gfCNCPoint1[2427] = {X 506.1982, Y 15.6317, Z -1.3333, A 0.000, B 0.000, C 0.000 }
gfCNCPoint1[2428] = {X 505.5600, Y 16.3119, Z -1.3333, A 0.000, B 0.000, C 0.000 }
gfCNCPoint1[2429] = {X 505.5599, Y 40.8749, Z -1.3333, A 0.000, B 0.000, C 0.000 }
gfCNCPoint1[2430] = {X 506.2050, Y 41.5641, Z -1.3333, A 0.000, B 0.000, C 0.000 }
gfCNCPoint1[2431] = {X 506.6882, Y 42.3750, Z -1.3333, A 0.000, B 0.000, C 0.000 }
gfCNCPoint1[2432] = {X 506.9873, Y 43.2704, Z -1.3333, A 0.000, B 0.000, C 0.000 }
gfCNCPoint1[2433] = {X 507.0885, Y 44.2089, Z -1.3333, A 0.000, B 0.000, C 0.000 }
gfCNCPoint1[2434] = {X 507.0885, Y 45.0000, Z -1.3333, A 0.000, B 0.000, C 0.000 }
gfCNCPoint1[2435] = {X 506.9782, Y 45.9791, Z -1.3333, A 0.000, B 0.000, C 0.000 }
gfCNCPoint1[2436] = {X 506.6528, Y 46.9091, Z -1.3333, A 0.000, B 0.000, C 0.000 }
gfCNCPoint1[2437] = {X 506.1285, Y 47.7434, Z -1.3333, A 0.000, B 0.000, C 0.000 }
gfCNCPoint1[2438] = {X 505.4318, Y 48.4401, Z -1.3333, A 0.000, B 0.000, C 0.000 }
gfCNCPoint1[2439] = {X 504.5976, Y 48.9643, Z -1.3333, A 0.000, B 0.000, C 0.000 }
gfCNCPoint1[2440] = {X 503.6676, Y 49.2897, Z -1.3333, A 0.000, B 0.000, C 0.000 }
gfCNCPoint1[2441] = {X 502.6885, Y 49.4000, Z -1.3333, A 0.000, B 0.000, C 0.000 }
gfCNCPoint1[2442] = {X 496.2450, Y 49.4000, Z -1.3333, A 0.000, B 0.000, C 0.000 }
gfCNCPoint1[2443] = {X 495.2659, Y 49.2897, Z -1.3333, A 0.000, B 0.000, C 0.000 }
gfCNCPoint1[2444] = {X 494.3359, Y 48.9643, Z -1.3333, A 0.000, B 0.000, C 0.000 }
gfCNCPoint1[2445] = {X 493.5017, Y 48.4400, Z -1.3333, A 0.000, B 0.000, C 0.000 }
gfCNCPoint1[2446] = {X 492.8049, Y 47.7433, Z -1.3333, A 0.000, B 0.000, C 0.000 }
gfCNCPoint1[2447] = {X 492.2807, Y 46.9091, Z -1.3333, A 0.000, B 0.000, C 0.000 }
gfCNCPoint1[2448] = {X 491.9553, Y 45.9790, Z -1.3333, A 0.000, B 0.000, C 0.000 }
gfCNCPoint1[2449] = {X 491.8450, Y 44.9999, Z -1.3333, A 0.000, B 0.000, C 0.000 }
gfCNCPoint1[2450] = {X 491.8454, Y 44.1483, Z -1.3333, A 0.000, B 0.000, C 0.000 }
gfCNCPoint1[2451] = {X 491.9559, Y 43.2275, Z -1.3333, A 0.000, B 0.000, C 0.000 }
gfCNCPoint1[2452] = {X 492.2568, Y 42.3503, Z -1.3333, A 0.000, B 0.000, C 0.000 }
gfCNCPoint1[2453] = {X 492.7349, Y 41.5556, Z -1.3333, A 0.000, B 0.000, C 0.000 }
gfCNCPoint1[2454] = {X 493.3690, Y 40.8789, Z -1.3333, A 0.000, B 0.000, C 0.000 }
gfCNCPoint1[2455] = {X 493.3690, Y 34.5538, Z -1.3333, A 0.000, B 0.000, C 0.000 }
gfCNCPoint1[2456] = {X 490.7720, Y 34.5538, Z -1.3333, A 0.000, B 0.000, C 0.000 }
gfCNCPoint1[2457] = {X 486.5265, Y 42.8211, Z -1.3333, A 0.000, B 0.000, C 0.000 }
gfCNCPoint1[2458] = {X 486.6945, Y 43.5060, Z -1.3333, A 0.000, B 0.000, C 0.000 }
gfCNCPoint1[2459] = {X 486.7510, Y 44.2089, Z -1.3333, A 0.000, B 0.000, C 0.000 }
gfCNCPoint1[2460] = {X 486.7510, Y 45.0000, Z -1.3333, A 0.000, B 0.000, C 0.000 }
gfCNCPoint1[2461] = {X 486.6407, Y 45.9791, Z -1.3333, A 0.000, B 0.000, C 0.000 }
gfCNCPoint1[2462] = {X 486.3153, Y 46.9091, Z -1.3333, A 0.000, B 0.000, C 0.000 }
gfCNCPoint1[2463] = {X 485.7911, Y 47.7434, Z -1.3333, A 0.000, B 0.000, C 0.000 }
gfCNCPoint1[2464] = {X 485.0944, Y 48.4401, Z -1.3333, A 0.000, B 0.000, C 0.000 }
gfCNCPoint1[2465] = {X 484.2601, Y 48.9643, Z -1.3333, A 0.000, B 0.000, C 0.000 }
gfCNCPoint1[2466] = {X 483.3301, Y 49.2897, Z -1.3333, A 0.000, B 0.000, C 0.000 }
gfCNCPoint1[2467] = {X 482.3510, Y 49.4000, Z -1.3333, A 0.000, B 0.000, C 0.000 }
gfCNCPoint1[2468] = {X 480.2695, Y 49.4000, Z -1.3333, A 0.000, B 0.000, C 0.000 }
gfCNCPoint1[2469] = {X 480.2695, Y 49.8800, Z -1.3333, A 0.000, B 0.000, C 0.000 }
gfCNCPoint1[2470] = {X 481.4067, Y 50.7435, Z -1.3333, A 0.000, B 0.000, C 0.000 }
gfCNCPoint1[2471] = {X 482.4044, Y 51.7649, Z -1.3333, A 0.000, B 0.000, C 0.000 }
gfCNCPoint1[2472] = {X 483.2411, Y 52.9219, Z -1.3333, A 0.000, B 0.000, C 0.000 }
gfCNCPoint1[2473] = {X 483.8615, Y 54.1044, Z -1.3333, A 0.000, B 0.000, C 0.000 }
gfCNCPoint1[2474] = {X 484.3133, Y 55.3610, Z -1.3333, A 0.000, B 0.000, C 0.000 }
gfCNCPoint1[2475] = {X 484.5879, Y 56.6678, Z -1.3333, A 0.000, B 0.000, C 0.000 }
gfCNCPoint1[2476] = {X 484.6800, Y 58.0000, Z -1.3333, A 0.000, B 0.000, C 0.000 }
gfCNCPoint1[2477] = {X 484.6797, Y 59.0140, Z -1.3333, A 0.000, B 0.000, C 0.000 }
gfCNCPoint1[2478] = {X 484.5592, Y 60.4586, Z -1.3333, A 0.000, B 0.000, C 0.000 }
gfCNCPoint1[2479] = {X 484.2243, Y 61.8690, Z -1.3333, A 0.000, B 0.000, C 0.000 }
gfCNCPoint1[2480] = {X 483.6826, Y 63.2136, Z -1.3333, A 0.000, B 0.000, C 0.000 }
gfCNCPoint1[2481] = {X 482.9462, Y 64.4622, Z -1.3333, A 0.000, B 0.000, C 0.000 }
gfCNCPoint1[2482] = {X 482.0316, Y 65.5868, Z -1.3333, A 0.000, B 0.000, C 0.000 }
gfCNCPoint1[2483] = {X 480.9593, Y 66.5623, Z -1.3333, A 0.000, B 0.000, C 0.000 }
gfCNCPoint1[2484] = {X 480.9596, Y 89.4452, Z -1.3333, A 0.000, B 0.000, C 0.000 }
gfCNCPoint1[2485] = {X 482.0591, Y 90.4472, Z -1.3333, A 0.000, B 0.000, C 0.000 }
gfCNCPoint1[2486] = {X 482.9917, Y 91.6063, Z -1.3333, A 0.000, B 0.000, C 0.000 }
gfCNCPoint1[2487] = {X 483.7350, Y 92.8949, Z -1.3333, A 0.000, B 0.000, C 0.000 }
gfCNCPoint1[2488] = {X 507.6820, Y 92.8949, Z -1.3333, A 0.000, B 0.000, C 0.000 }
gfCNCPoint1[2489] = {X 507.6820, Y 95.2949, Z -1.3333, A 0.000, B 0.000, C 0.000 }
gfCNCPoint1[2490] = {X 595.2965, Y 95.2949, Z -1.3333, A 0.000, B 0.000, C 0.000 }
gfCNCPoint1[2491] = {X 595.2965, Y 54.2000, Z -1.3333, A 0.000, B 0.000, C 0.000 }
gfCNCPoint1[2492] = {X 593.5565, Y 54.2000, Z -1.3333, A 0.000, B 0.000, C 0.000 }
gfCNCPoint1[2493] = {X 592.2403, Y 54.1053, Z -1.3333, A 0.000, B 0.000, C 0.000 }
gfCNCPoint1[2494] = {X 590.9511, Y 53.8233, Z -1.3333, A 0.000, B 0.000, C 0.000 }
gfCNCPoint1[2495] = {X 589.7155, Y 53.3598, Z -1.3333, A 0.000, B 0.000, C 0.000 }
gfCNCPoint1[2496] = {X 588.5589, Y 52.7242, Z -1.3333, A 0.000, B 0.000, C 0.000 }
gfCNCPoint1[2497] = {X 587.5052, Y 51.9297, Z -1.3333, A 0.000, B 0.000, C 0.000 }
gfCNCPoint1[2498] = {X 586.4956, Y 52.6955, Z -1.3333, A 0.000, B 0.000, C 0.000 }
gfCNCPoint1[2499] = {X 585.3903, Y 53.3153, Z -1.3333, A 0.000, B 0.000, C 0.000 }
gfCNCPoint1[2500] = {X 584.1375, Y 53.7999, Z -1.3333, A 0.000, B 0.000, C 0.000 }
gfCNCPoint1[2501] = {X 582.8276, Y 54.0969, Z -1.3333, A 0.000, B 0.000, C 0.000 }
gfCNCPoint1[2502] = {X 581.4884, Y 54.1999, Z -1.3333, A 0.000, B 0.000, C 0.000 }
gfCNCPoint1[2503] = {X 580.1485, Y 54.1069, Z -1.3333, A 0.000, B 0.000, C 0.000 }
gfCNCPoint1[2504] = {X 578.8364, Y 53.8198, Z -1.3333, A 0.000, B 0.000, C 0.000 }
gfCNCPoint1[2505] = {X 577.5801, Y 53.3447, Z -1.3333, A 0.000, B 0.000, C 0.000 }
gfCNCPoint1[2506] = {X 576.4063, Y 52.6917, Z -1.3333, A 0.000, B 0.000, C 0.000 }
gfCNCPoint1[2507] = {X 575.3401, Y 51.8748, Z -1.3333, A 0.000, B 0.000, C 0.000 }
gfCNCPoint1[2508] = {X 574.2798, Y 52.6879, Z -1.3333, A 0.000, B 0.000, C 0.000 }
gfCNCPoint1[2509] = {X 573.1128, Y 53.3388, Z -1.3333, A 0.000, B 0.000, C 0.000 }
gfCNCPoint1[2510] = {X 571.8638, Y 53.8139, Z -1.3333, A 0.000, B 0.000, C 0.000 }
gfCNCPoint1[2511] = {X 570.5592, Y 54.1030, Z -1.3333, A 0.000, B 0.000, C 0.000 }
gfCNCPoint1[2512] = {X 569.2264, Y 54.2000, Z -1.3333, A 0.000, B 0.000, C 0.000 }
gfCNCPoint1[2513] = {X 562.4443, Y 54.2000, Z -1.3333, A 0.000, B 0.000, C 0.000 }
gfCNCPoint1[2514] = {X 561.0051, Y 54.0867, Z -1.3333, A 0.000, B 0.000, C 0.000 }
gfCNCPoint1[2515] = {X 559.6013, Y 53.7497, Z -1.3333, A 0.000, B 0.000, C 0.000 }
gfCNCPoint1[2516] = {X 558.2676, Y 53.1973, Z -1.3333, A 0.000, B 0.000, C 0.000 }
gfCNCPoint1[2517] = {X 557.0367, Y 52.4430, Z -1.3333, A 0.000, B 0.000, C 0.000 }
gfCNCPoint1[2518] = {X 555.9389, Y 51.5054, Z -1.3333, A 0.000, B 0.000, C 0.000 }
gfCNCPoint1[2519] = {X 555.0013, Y 50.4076, Z -1.3333, A 0.000, B 0.000, C 0.000 }
gfCNCPoint1[2520] = {X 554.2470, Y 49.1767, Z -1.3333, A 0.000, B 0.000, C 0.000 }
gfCNCPoint1[2521] = {X 553.6946, Y 47.8430, Z -1.3333, A 0.000, B 0.000, C 0.000 }
gfCNCPoint1[2522] = {X 553.3576, Y 46.4392, Z -1.3333, A 0.000, B 0.000, C 0.000 }
gfCNCPoint1[2523] = {X 553.2443, Y 45.0000, Z -1.3333, A 0.000, B 0.000, C 0.000 }
gfCNCPoint1[2524] = {X 553.2443, Y 44.0589, Z -1.3333, A 0.000, B 0.000, C 0.000 }
gfCNCPoint1[2525] = {X 553.3454, Y 42.7230, Z -1.3333, A 0.000, B 0.000, C 0.000 }
gfCNCPoint1[2526] = {X 553.6387, Y 41.4159, Z -1.3333, A 0.000, B 0.000, C 0.000 }
gfCNCPoint1[2527] = {X 554.1179, Y 40.1649, Z -1.3333, A 0.000, B 0.000, C 0.000 }
gfCNCPoint1[2528] = {X 554.7730, Y 38.9963, Z -1.3333, A 0.000, B 0.000, C 0.000 }
gfCNCPoint1[2529] = {X 554.7730, Y 11.0125, Z -1.3333, A 0.000, B 0.000, C 0.000 }
gfCNCPoint1[2530] = {X 554.1225, Y 9.8568, Z -1.3333, A 0.000, B 0.000, C 0.000 }
gfCNCPoint1[2531] = {X 553.6449, Y 8.6195, Z -1.3333, A 0.000, B 0.000, C 0.000 }
gfCNCPoint1[2532] = {X 553.3503, Y 7.3264, Z -1.3333, A 0.000, B 0.000, C 0.000 }
gfCNCPoint1[2533] = {X 553.2446, Y 6.0043, Z -1.3333, A 0.000, B 0.000, C 0.000 }
gfCNCPoint1[2534] = {X 553.2443, Y 5.0000, Z -1.3333, A 0.000, B 0.000, C 0.000 }
gfCNCPoint1[2535] = {X 553.2455, Y 4.8525, Z -1.3333, A 0.000, B 0.000, C 0.000 }
gfCNCPoint1[2536] = {X 553.2490, Y 4.7051, Z -1.3333, A 0.000, B 0.000, C 0.000 }
gfCNCPoint1[2537] = {X 365.1858, Y 4.7051, Z -1.3333, A 0.000, B 0.000, C 0.000 }
gfCNCPoint1[2538] = {X 365.5690, Y 5.1220, Z -1.3333, A 0.000, B 0.000, C 0.000 }
gfCNCPoint1[2539] = {X 365.9422, Y 5.5478, Z -1.3333, A 0.000, B 0.000, C 0.000 }
gfCNCPoint1[2540] = {X 367.0635, Y 6.9475, Z -1.3333, A 0.000, B 0.000, C 0.000 }
gfCNCPoint1[2541] = {X 368.0917, Y 8.4168, Z -1.3333, A 0.000, B 0.000, C 0.000 }
gfCNCPoint1[2542] = {X 369.3445, Y 10.5369, Z -1.3333, A 0.000, B 0.000, C 0.000 }
gfCNCPoint1[2543] = {X 370.4040, Y 12.7600, Z -1.3333, A 0.000, B 0.000, C 0.000 }
gfCNCPoint1[2544] = {X 371.2616, Y 15.0684, Z -1.3333, A 0.000, B 0.000, C 0.000 }
gfCNCPoint1[2545] = {X 371.9107, Y 17.4439, Z -1.3333, A 0.000, B 0.000, C 0.000 }
gfCNCPoint1[2546] = {X 372.3638, Y 19.8385, Z -1.3333, A 0.000, B 0.000, C 0.000 }
gfCNCPoint1[2547] = {X 372.6472, Y 22.2590, Z -1.3333, A 0.000, B 0.000, C 0.000 }
gfCNCPoint1[2548] = {X 372.7595, Y 24.6935, Z -1.3333, A 0.000, B 0.000, C 0.000 }
gfCNCPoint1[2549] = {X 372.7001, Y 27.1298, Z -1.3333, A 0.000, B 0.000, C 0.000 }
gfCNCPoint1[2550] = {X 372.4694, Y 29.5560, Z -1.3333, A 0.000, B 0.000, C 0.000 }
gfCNCPoint1[2551] = {X 372.0685, Y 31.9598, Z -1.3333, A 0.000, B 0.000, C 0.000 }
gfCNCPoint1[2552] = {X 371.4818, Y 34.3169, Z -1.3333, A 0.000, B 0.000, C 0.000 }
gfCNCPoint1[2553] = {X 370.6892, Y 36.6130, Z -1.3333, A 0.000, B 0.000, C 0.000 }
gfCNCPoint1[2554] = {X 369.6968, Y 38.8301, Z -1.3333, A 0.000, B 0.000, C 0.000 }
gfCNCPoint1[2555] = {X 368.5125, Y 40.9509, Z -1.3333, A 0.000, B 0.000, C 0.000 }
gfCNCPoint1[2556] = {X 367.1454, Y 42.9587, Z -1.3333, A 0.000, B 0.000, C 0.000 }
gfCNCPoint1[2557] = {X 365.7525, Y 44.6742, Z -1.3333, A 0.000, B 0.000, C 0.000 }
gfCNCPoint1[2558] = {X 364.2142, Y 46.2608, Z -1.3333, A 0.000, B 0.000, C 0.000 }
gfCNCPoint1[2559] = {X 362.5426, Y 47.7061, Z -1.3333, A 0.000, B 0.000, C 0.000 }
gfCNCPoint1[2560] = {X 360.7505, Y 48.9991, Z -1.3333, A 0.000, B 0.000, C 0.000 }
gfCNCPoint1[2561] = {X 358.8518, Y 50.1297, Z -1.3333, A 0.000, B 0.000, C 0.000 }
gfCNCPoint1[2562] = {X 356.6370, Y 51.1396, Z -1.3333, A 0.000, B 0.000, C 0.000 }
gfCNCPoint1[2563] = {X 354.3363, Y 51.9345, Z -1.3333, A 0.000, B 0.000, C 0.000 }
gfCNCPoint1[2564] = {X 351.9704, Y 52.5073, Z -1.3333, A 0.000, B 0.000, C 0.000 }
gfCNCPoint1[2565] = {X 349.5608, Y 52.8527, Z -1.3333, A 0.000, B 0.000, C 0.000 }
gfCNCPoint1[2566] = {X 347.1293, Y 52.9676, Z -1.3333, A 0.000, B 0.000, C 0.000 }
gfCNCPoint1[2567] = {X 344.8095, Y 52.9250, Z -1.3333, A 0.000, B 0.000, C 0.000 }
gfCNCPoint1[2568] = {X 342.5021, Y 52.6816, Z -1.3333, A 0.000, B 0.000, C 0.000 }
gfCNCPoint1[2569] = {X 340.2244, Y 52.2394, Z -1.3333, A 0.000, B 0.000, C 0.000 }
gfCNCPoint1[2570] = {X 337.9936, Y 51.6015, Z -1.3333, A 0.000, B 0.000, C 0.000 }
gfCNCPoint1[2571] = {X 335.8264, Y 50.7729, Z -1.3333, A 0.000, B 0.000, C 0.000 }
gfCNCPoint1[2572] = {X 333.7392, Y 49.7597, Z -1.3333, A 0.000, B 0.000, C 0.000 }
gfCNCPoint1[2573] = {X 332.8270, Y 49.2213, Z -1.3333, A 0.000, B 0.000, C 0.000 }
gfCNCPoint1[2574] = {X 331.9366, Y 48.6477, Z -1.3333, A 0.000, B 0.000, C 0.000 }
gfCNCPoint1[2575] = {X 331.3044, Y 48.2095, Z -1.3333, A 0.000, B 0.000, C 0.000 }
gfCNCPoint1[2576] = {X 330.6849, Y 47.7536, Z -1.3333, A 0.000, B 0.000, C 0.000 }
gfCNCPoint1[2577] = {X 329.2349, Y 49.6661, Z -1.3333, A 0.000, B 0.000, C 0.000 }
gfCNCPoint1[2578] = {X 328.8833, Y 49.3953, Z -1.3333, A 0.000, B 0.000, C 0.000 }
gfCNCPoint1[2579] = {X 328.5358, Y 49.1193, Z -1.3333, A 0.000, B 0.000, C 0.000 }
gfCNCPoint1[2580] = {X 328.1287, Y 49.0395, Z -1.3333, A 0.000, B 0.000, C 0.000 }
gfCNCPoint1[2581] = {X 327.7253, Y 48.9423, Z -1.3333, A 0.000, B 0.000, C 0.000 }
gfCNCPoint1[2582] = {X 328.4958, Y 49.2715, Z -1.3333, A 0.000, B 0.000, C 0.000 }
gfCNCPoint1[2583] = {X 329.2349, Y 49.6661, Z -1.3333, A 0.000, B 0.000, C 0.000 }
gfCNCPoint1[2584] = {X 330.6849, Y 47.7536, Z -1.3333, A 0.000, B 0.000, C 0.000 }
gfCNCPoint1[2585] = {X 330.1044, Y 47.3009, Z -1.3333, A 0.000, B 0.000, C 0.000 }
gfCNCPoint1[2586] = {X 329.5364, Y 46.8326, Z -1.3333, A 0.000, B 0.000, C 0.000 }
gfCNCPoint1[2587] = {X 328.9325, Y 46.7522, Z -1.3333, A 0.000, B 0.000, C 0.000 }
gfCNCPoint1[2588] = {X 328.3374, Y 46.6216, Z -1.3333, A 0.000, B 0.000, C 0.000 }
gfCNCPoint1[2589] = {X 327.9789, Y 46.5172, Z -1.3333, A 0.000, B 0.000, C 0.000 }
gfCNCPoint1[2590] = {X 327.6263, Y 46.3944, Z -1.3333, A 0.000, B 0.000, C 0.000 }
gfCNCPoint1[2591] = {X 326.7320, Y 45.9864, Z -1.3333, A 0.000, B 0.000, C 0.000 }
gfCNCPoint1[2592] = {X 325.9009, Y 45.4616, Z -1.3333, A 0.000, B 0.000, C 0.000 }
gfCNCPoint1[2593] = {X 325.1480, Y 44.8296, Z -1.3333, A 0.000, B 0.000, C 0.000 }
gfCNCPoint1[2594] = {X 324.5140, Y 44.2115, Z -1.3333, A 0.000, B 0.000, C 0.000 }
gfCNCPoint1[2595] = {X 324.0475, Y 43.7117, Z -1.3333, A 0.000, B 0.000, C 0.000 }
gfCNCPoint1[2596] = {X 323.6300, Y 43.1703, Z -1.3333, A 0.000, B 0.000, C 0.000 }
gfCNCPoint1[2597] = {X 319.6957, Y 45.9200, Z -1.3333, A 0.000, B 0.000, C 0.000 }
gfCNCPoint1[2598] = {X 319.4780, Y 45.5976, Z -1.3333, A 0.000, B 0.000, C 0.000 }
gfCNCPoint1[2599] = {X 319.2708, Y 45.2683, Z -1.3333, A 0.000, B 0.000, C 0.000 }
gfCNCPoint1[2600] = {X 319.2514, Y 45.5948, Z -1.3333, A 0.000, B 0.000, C 0.000 }
gfCNCPoint1[2601] = {X 319.2174, Y 45.9200, Z -1.3333, A 0.000, B 0.000, C 0.000 }
gfCNCPoint1[2602] = {X 319.6957, Y 45.9200, Z -1.3333, A 0.000, B 0.000, C 0.000 }
gfCNCPoint1[2603] = {X 321.6628, Y 44.5452, Z -1.3333, A 0.000, B 0.000, C 0.000 }
gfCNCPoint1[2604] = {X 321.4884, Y 44.2868, Z -1.3333, A 0.000, B 0.000, C 0.000 }
gfCNCPoint1[2605] = {X 321.3224, Y 44.0230, Z -1.3333, A 0.000, B 0.000, C 0.000 }
gfCNCPoint1[2606] = {X 320.6715, Y 42.7462, Z -1.3333, A 0.000, B 0.000, C 0.000 }
gfCNCPoint1[2607] = {X 320.2162, Y 41.3874, Z -1.3333, A 0.000, B 0.000, C 0.000 }
gfCNCPoint1[2608] = {X 319.9665, Y 39.9762, Z -1.3333, A 0.000, B 0.000, C 0.000 }
gfCNCPoint1[2609] = {X 319.9279, Y 38.5436, Z -1.3333, A 0.000, B 0.000, C 0.000 }
gfCNCPoint1[2610] = {X 320.1013, Y 37.1210, Z -1.3333, A 0.000, B 0.000, C 0.000 }
gfCNCPoint1[2611] = {X 320.4293, Y 35.8933, Z -1.3333, A 0.000, B 0.000, C 0.000 }
gfCNCPoint1[2612] = {X 320.9152, Y 34.7191, Z -1.3333, A 0.000, B 0.000, C 0.000 }
gfCNCPoint1[2613] = {X 321.5508, Y 33.6186, Z -1.3333, A 0.000, B 0.000, C 0.000 }
gfCNCPoint1[2614] = {X 324.1369, Y 29.7518, Z -1.3333, A 0.000, B 0.000, C 0.000 }
gfCNCPoint1[2615] = {X 320.1470, Y 27.0834, Z -1.3333, A 0.000, B 0.000, C 0.000 }
gfCNCPoint1[2616] = {X 321.7941, Y 24.6207, Z -1.3333, A 0.000, B 0.000, C 0.000 }
gfCNCPoint1[2617] = {X 321.9845, Y 24.3430, Z -1.3333, A 0.000, B 0.000, C 0.000 }
gfCNCPoint1[2618] = {X 322.1814, Y 24.0697, Z -1.3333, A 0.000, B 0.000, C 0.000 }
gfCNCPoint1[2619] = {X 321.5380, Y 23.0772, Z -1.3333, A 0.000, B 0.000, C 0.000 }
gfCNCPoint1[2620] = {X 320.9777, Y 22.0355, Z -1.3333, A 0.000, B 0.000, C 0.000 }
gfCNCPoint1[2621] = {X 320.1471, Y 20.3268, Z -1.3333, A 0.000, B 0.000, C 0.000 }
gfCNCPoint1[2622] = {X 320.1470, Y 27.0834, Z -1.3333, A 0.000, B 0.000, C 0.000 }
gfCNCPoint1[2623] = {X 322.1420, Y 28.4176, Z -1.3333, A 0.000, B 0.000, C 0.000 }
gfCNCPoint1[2624] = {X 323.7890, Y 25.9549, Z -1.3333, A 0.000, B 0.000, C 0.000 }
gfCNCPoint1[2625] = {X 324.5064, Y 24.9899, Z -1.3333, A 0.000, B 0.000, C 0.000 }
gfCNCPoint1[2626] = {X 325.3162, Y 24.1010, Z -1.3333, A 0.000, B 0.000, C 0.000 }
gfCNCPoint1[2627] = {X 324.4812, Y 23.1413, Z -1.3333, A 0.000, B 0.000, C 0.000 }
gfCNCPoint1[2628] = {X 323.7518, Y 22.0990, Z -1.3333, A 0.000, B 0.000, C 0.000 }
gfCNCPoint1[2629] = {X 323.1360, Y 20.9859, Z -1.3333, A 0.000, B 0.000, C 0.000 }
gfCNCPoint1[2630] = {X 319.6151, Y 13.7428, Z -1.3333, A 0.000, B 0.000, C 0.000 }
gfCNCPoint1[2631] = {X 319.4387, Y 13.3633, Z -1.3333, A 0.000, B 0.000, C 0.000 }
gfCNCPoint1[2632] = {X 319.2755, Y 12.9779, Z -1.3333, A 0.000, B 0.000, C 0.000 }
gfCNCPoint1[2633] = {X 319.2755, Y 13.0353, Z -1.3333, A 0.000, B 0.000, C 0.000 }
gfCNCPoint1[2634] = {X 319.1697, Y 14.2160, Z -1.3333, A 0.000, B 0.000, C 0.000 }
gfCNCPoint1[2635] = {X 318.8737, Y 15.3639, Z -1.3333, A 0.000, B 0.000, C 0.000 }
gfCNCPoint1[2636] = {X 318.3952, Y 16.4486, Z -1.3333, A 0.000, B 0.000, C 0.000 }
gfCNCPoint1[2637] = {X 317.7471, Y 17.4412, Z -1.3333, A 0.000, B 0.000, C 0.000 }
gfCNCPoint1[2638] = {X 317.7469, Y 36.6552, Z -1.3333, A 0.000, B 0.000, C 0.000 }
gfCNCPoint1[2639] = {X 318.1562, Y 35.1230, Z -1.3333, A 0.000, B 0.000, C 0.000 }
gfCNCPoint1[2640] = {X 318.7627, Y 33.6577, Z -1.3333, A 0.000, B 0.000, C 0.000 }
gfCNCPoint1[2641] = {X 319.5559, Y 32.2844, Z -1.3333, A 0.000, B 0.000, C 0.000 }
gfCNCPoint1[2642] = {X 322.1420, Y 28.4176, Z -1.3333, A 0.000, B 0.000, C 0.000 }
gfCNCPoint1[2643] = {X 324.1369, Y 29.7518, Z -1.3333, A 0.000, B 0.000, C 0.000 }
gfCNCPoint1[2644] = {X 325.7840, Y 27.2892, Z -1.3333, A 0.000, B 0.000, C 0.000 }
gfCNCPoint1[2645] = {X 326.3588, Y 26.5158, Z -1.3333, A 0.000, B 0.000, C 0.000 }
gfCNCPoint1[2646] = {X 327.0077, Y 25.8035, Z -1.3333, A 0.000, B 0.000, C 0.000 }
gfCNCPoint1[2647] = {X 328.0707, Y 24.8904, Z -1.3333, A 0.000, B 0.000, C 0.000 }
gfCNCPoint1[2648] = {X 329.2543, Y 24.1403, Z -1.3333, A 0.000, B 0.000, C 0.000 }
gfCNCPoint1[2649] = {X 328.0859, Y 23.3667, Z -1.3333, A 0.000, B 0.000, C 0.000 }
gfCNCPoint1[2650] = {X 327.0414, Y 22.4326, Z -1.3333, A 0.000, B 0.000, C 0.000 }
gfCNCPoint1[2651] = {X 326.3723, Y 21.6635, Z -1.3333, A 0.000, B 0.000, C 0.000 }
gfCNCPoint1[2652] = {X 325.7878, Y 20.8284, Z -1.3333, A 0.000, B 0.000, C 0.000 }
gfCNCPoint1[2653] = {X 325.2944, Y 19.9364, Z -1.3333, A 0.000, B 0.000, C 0.000 }
gfCNCPoint1[2654] = {X 321.7736, Y 12.6936, Z -1.3333, A 0.000, B 0.000, C 0.000 }
gfCNCPoint1[2655] = {X 321.6322, Y 12.3894, Z -1.3333, A 0.000, B 0.000, C 0.000 }
gfCNCPoint1[2656] = {X 321.5015, Y 12.0806, Z -1.3333, A 0.000, B 0.000, C 0.000 }
gfCNCPoint1[2657] = {X 321.1058, Y 10.8774, Z -1.3333, A 0.000, B 0.000, C 0.000 }
gfCNCPoint1[2658] = {X 320.8706, Y 9.6328, Z -1.3333, A 0.000, B 0.000, C 0.000 }
gfCNCPoint1[2659] = {X 320.7999, Y 8.3682, Z -1.3333, A 0.000, B 0.000, C 0.000 }
gfCNCPoint1[2660] = {X 320.8950, Y 7.1051, Z -1.3333, A 0.000, B 0.000, C 0.000 }
gfCNCPoint1[2661] = {X 298.7842, Y 7.1051, Z -1.3333, A 0.000, B 0.000, C 0.000 }
gfCNCPoint1[2662] = {X 298.7842, Y 9.5051, Z -1.3333, A 0.000, B 0.000, C 0.000 }
gfCNCPoint1[2663] = {X 297.8292, Y 9.5051, Z -1.3333, A 0.000, B 0.000, C 0.000 }
gfCNCPoint1[2664] = {X 298.1372, Y 10.4756, Z -1.3333, A 0.000, B 0.000, C 0.000 }
gfCNCPoint1[2665] = {X 298.3067, Y 11.4795, Z -1.3333, A 0.000, B 0.000, C 0.000 }
gfCNCPoint1[2666] = {X 298.4762, Y 10.4756, Z -1.3333, A 0.000, B 0.000, C 0.000 }
gfCNCPoint1[2667] = {X 298.7842, Y 9.5051, Z -1.3333, A 0.000, B 0.000, C 0.000 }
gfCNCPoint1[2668] = {X 298.7842, Y 7.1051, Z -1.3333, A 0.000, B 0.000, C 0.000 }
gfCNCPoint1[2669] = {X 233.3055, Y 7.1051, Z -1.3333, A 0.000, B 0.000, C 0.000 }
gfCNCPoint1[2670] = {X 233.3055, Y 11.9051, Z -1.3333, A 0.000, B 0.000, C 0.000 }
gfCNCPoint1[2671] = {X 233.1564, Y 11.9051, Z -1.3333, A 0.000, B 0.000, C 0.000 }
gfCNCPoint1[2672] = {X 233.1595, Y 12.0461, Z -1.3333, A 0.000, B 0.000, C 0.000 }
gfCNCPoint1[2673] = {X 233.1605, Y 12.1872, Z -1.3333, A 0.000, B 0.000, C 0.000 }
gfCNCPoint1[2674] = {X 233.2324, Y 12.0458, Z -1.3333, A 0.000, B 0.000, C 0.000 }
gfCNCPoint1[2675] = {X 233.3055, Y 11.9051, Z -1.3333, A 0.000, B 0.000, C 0.000 }
gfCNCPoint1[2676] = {X 233.3055, Y 9.5051, Z -1.3333, A 0.000, B 0.000, C 0.000 }
gfCNCPoint1[2677] = {X 230.2486, Y 9.5051, Z -1.3333, A 0.000, B 0.000, C 0.000 }
gfCNCPoint1[2678] = {X 230.6107, Y 10.7178, Z -1.3333, A 0.000, B 0.000, C 0.000 }
gfCNCPoint1[2679] = {X 230.7574, Y 11.9750, Z -1.3333, A 0.000, B 0.000, C 0.000 }
gfCNCPoint1[2680] = {X 230.7597, Y 12.0809, Z -1.3333, A 0.000, B 0.000, C 0.000 }
gfCNCPoint1[2681] = {X 230.7605, Y 12.1868, Z -1.3333, A 0.000, B 0.000, C 0.000 }
gfCNCPoint1[2682] = {X 230.7602, Y 13.0462, Z -1.3333, A 0.000, B 0.000, C 0.000 }
gfCNCPoint1[2683] = {X 230.6531, Y 14.2240, Z -1.3333, A 0.000, B 0.000, C 0.000 }
gfCNCPoint1[2684] = {X 230.3567, Y 15.3689, Z -1.3333, A 0.000, B 0.000, C 0.000 }
gfCNCPoint1[2685] = {X 229.8788, Y 16.4507, Z -1.3333, A 0.000, B 0.000, C 0.000 }
gfCNCPoint1[2686] = {X 229.2321, Y 17.4409, Z -1.3333, A 0.000, B 0.000, C 0.000 }
gfCNCPoint1[2687] = {X 229.2324, Y 25.8394, Z -1.3333, A 0.000, B 0.000, C 0.000 }
gfCNCPoint1[2688] = {X 231.6324, Y 25.8393, Z -1.3333, A 0.000, B 0.000, C 0.000 }
gfCNCPoint1[2689] = {X 231.6329, Y 38.9895, Z -1.3333, A 0.000, B 0.000, C 0.000 }
gfCNCPoint1[2690] = {X 231.6440, Y 39.0069, Z -1.3333, A 0.000, B 0.000, C 0.000 }
gfCNCPoint1[2691] = {X 232.3931, Y 37.9855, Z -1.3333, A 0.000, B 0.000, C 0.000 }
gfCNCPoint1[2692] = {X 233.2692, Y 37.0706, Z -1.3333, A 0.000, B 0.000, C 0.000 }
gfCNCPoint1[2693] = {X 234.2573, Y 36.2780, Z -1.3333, A 0.000, B 0.000, C 0.000 }
gfCNCPoint1[2694] = {X 235.5699, Y 33.7088, Z -1.3333, A 0.000, B 0.000, C 0.000 }
gfCNCPoint1[2695] = {X 234.4293, Y 32.2848, Z -1.3333, A 0.000, B 0.000, C 0.000 }
gfCNCPoint1[2696] = {X 233.4512, Y 30.7447, Z -1.3333, A 0.000, B 0.000, C 0.000 }
gfCNCPoint1[2697] = {X 232.6471, Y 29.1070, Z -1.3333, A 0.000, B 0.000, C 0.000 }
gfCNCPoint1[2698] = {X 232.0268, Y 27.3912, Z -1.3333, A 0.000, B 0.000, C 0.000 }
gfCNCPoint1[2699] = {X 231.8154, Y 26.6188, Z -1.3333, A 0.000, B 0.000, C 0.000 }
gfCNCPoint1[2700] = {X 231.6324, Y 25.8393, Z -1.3333, A 0.000, B 0.000, C 0.000 }
gfCNCPoint1[2701] = {X 229.2324, Y 25.8394, Z -1.3333, A 0.000, B 0.000, C 0.000 }
gfCNCPoint1[2702] = {X 229.2329, Y 39.7469, Z -1.3333, A 0.000, B 0.000, C 0.000 }
gfCNCPoint1[2703] = {X 229.4328, Y 40.0173, Z -1.3333, A 0.000, B 0.000, C 0.000 }
gfCNCPoint1[2704] = {X 229.6200, Y 40.2966, Z -1.3333, A 0.000, B 0.000, C 0.000 }
gfCNCPoint1[2705] = {X 230.1055, Y 41.1910, Z -1.3333, A 0.000, B 0.000, C 0.000 }
gfCNCPoint1[2706] = {X 230.4616, Y 42.1443, Z -1.3333, A 0.000, B 0.000, C 0.000 }
gfCNCPoint1[2707] = {X 230.6813, Y 43.1379, Z -1.3333, A 0.000, B 0.000, C 0.000 }
gfCNCPoint1[2708] = {X 230.7603, Y 44.1524, Z -1.3333, A 0.000, B 0.000, C 0.000 }
gfCNCPoint1[2709] = {X 230.7605, Y 45.0000, Z -1.3333, A 0.000, B 0.000, C 0.000 }
gfCNCPoint1[2710] = {X 230.7459, Y 45.4609, Z -1.3333, A 0.000, B 0.000, C 0.000 }
gfCNCPoint1[2711] = {X 230.7021, Y 45.9200, Z -1.3333, A 0.000, B 0.000, C 0.000 }
gfCNCPoint1[2712] = {X 232.5859, Y 45.9200, Z -1.3333, A 0.000, B 0.000, C 0.000 }
gfCNCPoint1[2713] = {X 232.5421, Y 45.4609, Z -1.3333, A 0.000, B 0.000, C 0.000 }
gfCNCPoint1[2714] = {X 232.5275, Y 45.0000, Z -1.3333, A 0.000, B 0.000, C 0.000 }
gfCNCPoint1[2715] = {X 232.5275, Y 44.2090, Z -1.3333, A 0.000, B 0.000, C 0.000 }
gfCNCPoint1[2716] = {X 232.6006, Y 43.1799, Z -1.3333, A 0.000, B 0.000, C 0.000 }
gfCNCPoint1[2717] = {X 232.8184, Y 42.1714, Z -1.3333, A 0.000, B 0.000, C 0.000 }
gfCNCPoint1[2718] = {X 233.1766, Y 41.2038, Z -1.3333, A 0.000, B 0.000, C 0.000 }
gfCNCPoint1[2719] = {X 233.6680, Y 40.2966, Z -1.3333, A 0.000, B 0.000, C 0.000 }
gfCNCPoint1[2720] = {X 234.3527, Y 39.3876, Z -1.3333, A 0.000, B 0.000, C 0.000 }
gfCNCPoint1[2721] = {X 235.1707, Y 38.5964, Z -1.3333, A 0.000, B 0.000, C 0.000 }
gfCNCPoint1[2722] = {X 236.1021, Y 37.9424, Z -1.3333, A 0.000, B 0.000, C 0.000 }
gfCNCPoint1[2723] = {X 238.5004, Y 33.2478, Z -1.3333, A 0.000, B 0.000, C 0.000 }
gfCNCPoint1[2724] = {X 237.3869, Y 32.1402, Z -1.3333, A 0.000, B 0.000, C 0.000 }
gfCNCPoint1[2725] = {X 236.4017, Y 30.9169, Z -1.3333, A 0.000, B 0.000, C 0.000 }
gfCNCPoint1[2726] = {X 235.5569, Y 29.5929, Z -1.3333, A 0.000, B 0.000, C 0.000 }
gfCNCPoint1[2727] = {X 234.8627, Y 28.1840, Z -1.3333, A 0.000, B 0.000, C 0.000 }
gfCNCPoint1[2728] = {X 234.3274, Y 26.7074, Z -1.3333, A 0.000, B 0.000, C 0.000 }
gfCNCPoint1[2729] = {X 234.1404, Y 26.0237, Z -1.3333, A 0.000, B 0.000, C 0.000 }
gfCNCPoint1[2730] = {X 233.9785, Y 25.3335, Z -1.3333, A 0.000, B 0.000, C 0.000 }
gfCNCPoint1[2731] = {X 233.6677, Y 23.4469, Z -1.3333, A 0.000, B 0.000, C 0.000 }
gfCNCPoint1[2732] = {X 233.5433, Y 21.5390, Z -1.3333, A 0.000, B 0.000, C 0.000 }
gfCNCPoint1[2733] = {X 233.6063, Y 19.6280, Z -1.3333, A 0.000, B 0.000, C 0.000 }
gfCNCPoint1[2734] = {X 233.8562, Y 17.7323, Z -1.3333, A 0.000, B 0.000, C 0.000 }
gfCNCPoint1[2735] = {X 234.2907, Y 15.8703, Z -1.3333, A 0.000, B 0.000, C 0.000 }
gfCNCPoint1[2736] = {X 234.7361, Y 14.5437, Z -1.3333, A 0.000, B 0.000, C 0.000 }
gfCNCPoint1[2737] = {X 235.3048, Y 13.2651, Z -1.3333, A 0.000, B 0.000, C 0.000 }
gfCNCPoint1[2738] = {X 235.3667, Y 13.1434, Z -1.3333, A 0.000, B 0.000, C 0.000 }
gfCNCPoint1[2739] = {X 235.4296, Y 13.0223, Z -1.3333, A 0.000, B 0.000, C 0.000 }
gfCNCPoint1[2740] = {X 236.1709, Y 11.7671, Z -1.3333, A 0.000, B 0.000, C 0.000 }
gfCNCPoint1[2741] = {X 237.0321, Y 10.5909, Z -1.3333, A 0.000, B 0.000, C 0.000 }
gfCNCPoint1[2742] = {X 238.0047, Y 9.5051, Z -1.3333, A 0.000, B 0.000, C 0.000 }
gfCNCPoint1[2743] = {X 233.3055, Y 9.5051, Z -1.3333, A 0.000, B 0.000, C 0.000 }
gfCNCPoint1[2744] = {X 233.3055, Y 7.1051, Z -1.3333, A 0.000, B 0.000, C 0.000 }
gfCNCPoint1[2745] = {X 207.3611, Y 7.1051, Z -1.3333, A 0.000, B 0.000, C 0.000 }
gfCNCPoint1[2746] = {X 207.3611, Y 11.9051, Z -1.3333, A 0.000, B 0.000, C 0.000 }
gfCNCPoint1[2747] = {X 205.8549, Y 11.9051, Z -1.3333, A 0.000, B 0.000, C 0.000 }
gfCNCPoint1[2748] = {X 206.6100, Y 13.3411, Z -1.3333, A 0.000, B 0.000, C 0.000 }
gfCNCPoint1[2749] = {X 207.2356, Y 14.8379, Z -1.3333, A 0.000, B 0.000, C 0.000 }
gfCNCPoint1[2750] = {X 207.7967, Y 16.7109, Z -1.3333, A 0.000, B 0.000, C 0.000 }
gfCNCPoint1[2751] = {X 208.1757, Y 18.6291, Z -1.3333, A 0.000, B 0.000, C 0.000 }
gfCNCPoint1[2752] = {X 208.3692, Y 20.5747, Z -1.3333, A 0.000, B 0.000, C 0.000 }
gfCNCPoint1[2753] = {X 208.3753, Y 22.5299, Z -1.3333, A 0.000, B 0.000, C 0.000 }
gfCNCPoint1[2754] = {X 208.1941, Y 24.4767, Z -1.3333, A 0.000, B 0.000, C 0.000 }
gfCNCPoint1[2755] = {X 207.8272, Y 26.3972, Z -1.3333, A 0.000, B 0.000, C 0.000 }
gfCNCPoint1[2756] = {X 207.3604, Y 28.0094, Z -1.3333, A 0.000, B 0.000, C 0.000 }
gfCNCPoint1[2757] = {X 206.7372, Y 29.5678, Z -1.3333, A 0.000, B 0.000, C 0.000 }
gfCNCPoint1[2758] = {X 205.9639, Y 31.0574, Z -1.3333, A 0.000, B 0.000, C 0.000 }
gfCNCPoint1[2759] = {X 206.0462, Y 31.2160, Z -1.3333, A 0.000, B 0.000, C 0.000 }
gfCNCPoint1[2760] = {X 206.1255, Y 31.3761, Z -1.3333, A 0.000, B 0.000, C 0.000 }
gfCNCPoint1[2761] = {X 208.8862, Y 37.0796, Z -1.3333, A 0.000, B 0.000, C 0.000 }
gfCNCPoint1[2762] = {X 208.8862, Y 18.1998, Z -1.3333, A 0.000, B 0.000, C 0.000 }
gfCNCPoint1[2763] = {X 208.2337, Y 17.0034, Z -1.3333, A 0.000, B 0.000, C 0.000 }
gfCNCPoint1[2764] = {X 207.7556, Y 15.7272, Z -1.3333, A 0.000, B 0.000, C 0.000 }
gfCNCPoint1[2765] = {X 207.4615, Y 14.3965, Z -1.3333, A 0.000, B 0.000, C 0.000 }
gfCNCPoint1[2766] = {X 207.3572, Y 13.0378, Z -1.3333, A 0.000, B 0.000, C 0.000 }
gfCNCPoint1[2767] = {X 207.3570, Y 12.1868, Z -1.3333, A 0.000, B 0.000, C 0.000 }
gfCNCPoint1[2768] = {X 207.3580, Y 12.0459, Z -1.3333, A 0.000, B 0.000, C 0.000 }
gfCNCPoint1[2769] = {X 207.3611, Y 11.9051, Z -1.3333, A 0.000, B 0.000, C 0.000 }
gfCNCPoint1[2770] = {X 207.3611, Y 9.5051, Z -1.3333, A 0.000, B 0.000, C 0.000 }
gfCNCPoint1[2771] = {X 200.9060, Y 9.5051, Z -1.3333, A 0.000, B 0.000, C 0.000 }
gfCNCPoint1[2772] = {X 201.9793, Y 10.6138, Z -1.3333, A 0.000, B 0.000, C 0.000 }
gfCNCPoint1[2773] = {X 202.9410, Y 11.8207, Z -1.3333, A 0.000, B 0.000, C 0.000 }
gfCNCPoint1[2774] = {X 203.7820, Y 13.1146, Z -1.3333, A 0.000, B 0.000, C 0.000 }
gfCNCPoint1[2775] = {X 204.4353, Y 14.3564, Z -1.3333, A 0.000, B 0.000, C 0.000 }
gfCNCPoint1[2776] = {X 204.9774, Y 15.6507, Z -1.3333, A 0.000, B 0.000, C 0.000 }
gfCNCPoint1[2777] = {X 205.5500, Y 17.6374, Z -1.3333, A 0.000, B 0.000, C 0.000 }
gfCNCPoint1[2778] = {X 205.8909, Y 19.6766, Z -1.3333, A 0.000, B 0.000, C 0.000 }
gfCNCPoint1[2779] = {X 205.9954, Y 21.7416, Z -1.3333, A 0.000, B 0.000, C 0.000 }
gfCNCPoint1[2780] = {X 205.8622, Y 23.8048, Z -1.3333, A 0.000, B 0.000, C 0.000 }
gfCNCPoint1[2781] = {X 205.4930, Y 25.8392, Z -1.3333, A 0.000, B 0.000, C 0.000 }
gfCNCPoint1[2782] = {X 205.0921, Y 27.2252, Z -1.3333, A 0.000, B 0.000, C 0.000 }
gfCNCPoint1[2783] = {X 204.5567, Y 28.5652, Z -1.3333, A 0.000, B 0.000, C 0.000 }
gfCNCPoint1[2784] = {X 203.8921, Y 29.8459, Z -1.3333, A 0.000, B 0.000, C 0.000 }
gfCNCPoint1[2785] = {X 203.1048, Y 31.0551, Z -1.3333, A 0.000, B 0.000, C 0.000 }
gfCNCPoint1[2786] = {X 203.5730, Y 31.7144, Z -1.3333, A 0.000, B 0.000, C 0.000 }
gfCNCPoint1[2787] = {X 203.9653, Y 32.4217, Z -1.3333, A 0.000, B 0.000, C 0.000 }
gfCNCPoint1[2788] = {X 206.9865, Y 38.6634, Z -1.3333, A 0.000, B 0.000, C 0.000 }
gfCNCPoint1[2789] = {X 207.4240, Y 39.8017, Z -1.3333, A 0.000, B 0.000, C 0.000 }
gfCNCPoint1[2790] = {X 207.6653, Y 40.9971, Z -1.3333, A 0.000, B 0.000, C 0.000 }
gfCNCPoint1[2791] = {X 207.7038, Y 42.2159, Z -1.3333, A 0.000, B 0.000, C 0.000 }
gfCNCPoint1[2792] = {X 207.5382, Y 43.4241, Z -1.3333, A 0.000, B 0.000, C 0.000 }
gfCNCPoint1[2793] = {X 207.1733, Y 44.5877, Z -1.3333, A 0.000, B 0.000, C 0.000 }
gfCNCPoint1[2794] = {X 206.6193, Y 45.6741, Z -1.3333, A 0.000, B 0.000, C 0.000 }
gfCNCPoint1[2795] = {X 205.8917, Y 46.6527, Z -1.3333, A 0.000, B 0.000, C 0.000 }
gfCNCPoint1[2796] = {X 205.0110, Y 47.4962, Z -1.3333, A 0.000, B 0.000, C 0.000 }
gfCNCPoint1[2797] = {X 204.4723, Y 47.9317, Z -1.3333, A 0.000, B 0.000, C 0.000 }
gfCNCPoint1[2798] = {X 203.5887, Y 48.5429, Z -1.3333, A 0.000, B 0.000, C 0.000 }
gfCNCPoint1[2799] = {X 202.6249, Y 49.0177, Z -1.3333, A 0.000, B 0.000, C 0.000 }
gfCNCPoint1[2800] = {X 201.4908, Y 49.3717, Z -1.3333, A 0.000, B 0.000, C 0.000 }
gfCNCPoint1[2801] = {X 200.3142, Y 49.5370, Z -1.3333, A 0.000, B 0.000, C 0.000 }
gfCNCPoint1[2802] = {X 199.1265, Y 49.5092, Z -1.3333, A 0.000, B 0.000, C 0.000 }
gfCNCPoint1[2803] = {X 198.4543, Y 49.8548, Z -1.3333, A 0.000, B 0.000, C 0.000 }
gfCNCPoint1[2804] = {X 197.7738, Y 50.1840, Z -1.3333, A 0.000, B 0.000, C 0.000 }
gfCNCPoint1[2805] = {X 199.8113, Y 54.5301, Z -1.3333, A 0.000, B 0.000, C 0.000 }
gfCNCPoint1[2806] = {X 197.9066, Y 55.3565, Z -1.3333, A 0.000, B 0.000, C 0.000 }
gfCNCPoint1[2807] = {X 195.9573, Y 56.0711, Z -1.3333, A 0.000, B 0.000, C 0.000 }
gfCNCPoint1[2808] = {X 195.3265, Y 56.2889, Z -1.3333, A 0.000, B 0.000, C 0.000 }
gfCNCPoint1[2809] = {X 195.3581, Y 56.6331, Z -1.3333, A 0.000, B 0.000, C 0.000 }
gfCNCPoint1[2810] = {X 195.3825, Y 56.9779, Z -1.3333, A 0.000, B 0.000, C 0.000 }
gfCNCPoint1[2811] = {X 199.6723, Y 61.6596, Z -1.3333, A 0.000, B 0.000, C 0.000 }
gfCNCPoint1[2812] = {X 199.5095, Y 60.3409, Z -1.3333, A 0.000, B 0.000, C 0.000 }
gfCNCPoint1[2813] = {X 199.4510, Y 59.0136, Z -1.3333, A 0.000, B 0.000, C 0.000 }
gfCNCPoint1[2814] = {X 199.4508, Y 58.0000, Z -1.3333, A 0.000, B 0.000, C 0.000 }
gfCNCPoint1[2815] = {X 199.5412, Y 56.2557, Z -1.3333, A 0.000, B 0.000, C 0.000 }
gfCNCPoint1[2816] = {X 199.8113, Y 54.5301, Z -1.3333, A 0.000, B 0.000, C 0.000 }
gfCNCPoint1[2817] = {X 198.7926, Y 52.3571, Z -1.3333, A 0.000, B 0.000, C 0.000 }
gfCNCPoint1[2818] = {X 197.0101, Y 53.1303, Z -1.3333, A 0.000, B 0.000, C 0.000 }
gfCNCPoint1[2819] = {X 195.1856, Y 53.7985, Z -1.3333, A 0.000, B 0.000, C 0.000 }
gfCNCPoint1[2820] = {X 194.5578, Y 54.0153, Z -1.3333, A 0.000, B 0.000, C 0.000 }
gfCNCPoint1[2821] = {X 193.5844, Y 54.3097, Z -1.3333, A 0.000, B 0.000, C 0.000 }
gfCNCPoint1[2822] = {X 192.6011, Y 54.5688, Z -1.3333, A 0.000, B 0.000, C 0.000 }
gfCNCPoint1[2823] = {X 192.9067, Y 56.2447, Z -1.3333, A 0.000, B 0.000, C 0.000 }
gfCNCPoint1[2824] = {X 193.0134, Y 57.9448, Z -1.3333, A 0.000, B 0.000, C 0.000 }
gfCNCPoint1[2825] = {X 210.3933, Y 76.9128, Z -1.3333, A 0.000, B 0.000, C 0.000 }
gfCNCPoint1[2826] = {X 212.1628, Y 75.2914, Z -1.3333, A 0.000, B 0.000, C 0.000 }
gfCNCPoint1[2827] = {X 215.1993, Y 78.6053, Z -1.3333, A 0.000, B 0.000, C 0.000 }
gfCNCPoint1[2828] = {X 218.3298, Y 76.5996, Z -1.3333, A 0.000, B 0.000, C 0.000 }
gfCNCPoint1[2829] = {X 216.9961, Y 76.0762, Z -1.3333, A 0.000, B 0.000, C 0.000 }
gfCNCPoint1[2830] = {X 216.3783, Y 75.8845, Z -1.3333, A 0.000, B 0.000, C 0.000 }
gfCNCPoint1[2831] = {X 215.7364, Y 75.8036, Z -1.3333, A 0.000, B 0.000, C 0.000 }
gfCNCPoint1[2832] = {X 213.9359, Y 75.6433, Z -1.3333, A 0.000, B 0.000, C 0.000 }
gfCNCPoint1[2833] = {X 212.1628, Y 75.2914, Z -1.3333, A 0.000, B 0.000, C 0.000 }
gfCNCPoint1[2834] = {X 210.3933, Y 76.9128, Z -1.3333, A 0.000, B 0.000, C 0.000 }
gfCNCPoint1[2835] = {X 214.7938, Y 81.7153, Z -1.3333, A 0.000, B 0.000, C 0.000 }
gfCNCPoint1[2836] = {X 223.5843, Y 76.0836, Z -1.3333, A 0.000, B 0.000, C 0.000 }
gfCNCPoint1[2837] = {X 217.8854, Y 73.8470, Z -1.3333, A 0.000, B 0.000, C 0.000 }
gfCNCPoint1[2838] = {X 216.8736, Y 73.5361, Z -1.3333, A 0.000, B 0.000, C 0.000 }
gfCNCPoint1[2839] = {X 215.8232, Y 73.4052, Z -1.3333, A 0.000, B 0.000, C 0.000 }
gfCNCPoint1[2840] = {X 214.2776, Y 73.2678, Z -1.3333, A 0.000, B 0.000, C 0.000 }
gfCNCPoint1[2841] = {X 212.7554, Y 72.9657, Z -1.3333, A 0.000, B 0.000, C 0.000 }
gfCNCPoint1[2842] = {X 211.1566, Y 72.4581, Z -1.3333, A 0.000, B 0.000, C 0.000 }
gfCNCPoint1[2843] = {X 209.6273, Y 71.7689, Z -1.3333, A 0.000, B 0.000, C 0.000 }
gfCNCPoint1[2844] = {X 208.1879, Y 70.9075, Z -1.3333, A 0.000, B 0.000, C 0.000 }
gfCNCPoint1[2845] = {X 206.8577, Y 69.8854, Z -1.3333, A 0.000, B 0.000, C 0.000 }
gfCNCPoint1[2846] = {X 205.6547, Y 68.7163, Z -1.3333, A 0.000, B 0.000, C 0.000 }
gfCNCPoint1[2847] = {X 204.5950, Y 67.4159, Z -1.3333, A 0.000, B 0.000, C 0.000 }
gfCNCPoint1[2848] = {X 203.6928, Y 66.0018, Z -1.3333, A 0.000, B 0.000, C 0.000 }
gfCNCPoint1[2849] = {X 202.9602, Y 64.4927, Z -1.3333, A 0.000, B 0.000, C 0.000 }
gfCNCPoint1[2850] = {X 202.4071, Y 62.9091, Z -1.3333, A 0.000, B 0.000, C 0.000 }
gfCNCPoint1[2851] = {X 202.0408, Y 61.2721, Z -1.3333, A 0.000, B 0.000, C 0.000 }
gfCNCPoint1[2852] = {X 201.9014, Y 60.1434, Z -1.3333, A 0.000, B 0.000, C 0.000 }
gfCNCPoint1[2853] = {X 201.8510, Y 59.0073, Z -1.3333, A 0.000, B 0.000, C 0.000 }
gfCNCPoint1[2854] = {X 201.8508, Y 58.0000, Z -1.3333, A 0.000, B 0.000, C 0.000 }
gfCNCPoint1[2855] = {X 201.9283, Y 56.5037, Z -1.3333, A 0.000, B 0.000, C 0.000 }
gfCNCPoint1[2856] = {X 202.1600, Y 55.0235, Z -1.3333, A 0.000, B 0.000, C 0.000 }
gfCNCPoint1[2857] = {X 202.4969, Y 53.7228, Z -1.3333, A 0.000, B 0.000, C 0.000 }
gfCNCPoint1[2858] = {X 202.9529, Y 52.4590, Z -1.3333, A 0.000, B 0.000, C 0.000 }
gfCNCPoint1[2859] = {X 203.5241, Y 51.2429, Z -1.3333, A 0.000, B 0.000, C 0.000 }
gfCNCPoint1[2860] = {X 202.2650, Y 51.6541, Z -1.3333, A 0.000, B 0.000, C 0.000 }
gfCNCPoint1[2861] = {X 200.9616, Y 51.8900, Z -1.3333, A 0.000, B 0.000, C 0.000 }
gfCNCPoint1[2862] = {X 199.6382, Y 51.9460, Z -1.3333, A 0.000, B 0.000, C 0.000 }
gfCNCPoint1[2863] = {X 199.2168, Y 52.1545, Z -1.3333, A 0.000, B 0.000, C 0.000 }
gfCNCPoint1[2864] = {X 198.7926, Y 52.3571, Z -1.3333, A 0.000, B 0.000, C 0.000 }
gfCNCPoint1[2865] = {X 197.7738, Y 50.1840, Z -1.3333, A 0.000, B 0.000, C 0.000 }
gfCNCPoint1[2866] = {X 196.1132, Y 50.9041, Z -1.3333, A 0.000, B 0.000, C 0.000 }
gfCNCPoint1[2867] = {X 194.4134, Y 51.5260, Z -1.3333, A 0.000, B 0.000, C 0.000 }
gfCNCPoint1[2868] = {X 193.8217, Y 51.7310, Z -1.3333, A 0.000, B 0.000, C 0.000 }
gfCNCPoint1[2869] = {X 192.9311, Y 52.0003, Z -1.3333, A 0.000, B 0.000, C 0.000 }
gfCNCPoint1[2870] = {X 192.0315, Y 52.2374, Z -1.3333, A 0.000, B 0.000, C 0.000 }
gfCNCPoint1[2871] = {X 190.7254, Y 52.5209, Z -1.3333, A 0.000, B 0.000, C 0.000 }
gfCNCPoint1[2872] = {X 189.4065, Y 52.7364, Z -1.3333, A 0.000, B 0.000, C 0.000 }
gfCNCPoint1[2873] = {X 189.9015, Y 53.9141, Z -1.3333, A 0.000, B 0.000, C 0.000 }
gfCNCPoint1[2874] = {X 190.2695, Y 55.1375, Z -1.3333, A 0.000, B 0.000, C 0.000 }
gfCNCPoint1[2875] = {X 190.5272, Y 56.5585, Z -1.3333, A 0.000, B 0.000, C 0.000 }
gfCNCPoint1[2876] = {X 190.6135, Y 58.0000, Z -1.3333, A 0.000, B 0.000, C 0.000 }
gfCNCPoint1[2877] = {X 190.6132, Y 58.8779, Z -1.3333, A 0.000, B 0.000, C 0.000 }
gfCNCPoint1[2878] = {X 214.3883, Y 84.8254, Z -1.3333, A 0.000, B 0.000, C 0.000 }
gfCNCPoint1[2879] = {X 228.8388, Y 75.5676, Z -1.3333, A 0.000, B 0.000, C 0.000 }
gfCNCPoint1[2880] = {X 218.7726, Y 71.6170, Z -1.3333, A 0.000, B 0.000, C 0.000 }
gfCNCPoint1[2881] = {X 217.8439, Y 71.3035, Z -1.3333, A 0.000, B 0.000, C 0.000 }
gfCNCPoint1[2882] = {X 216.8852, Y 71.0992, Z -1.3333, A 0.000, B 0.000, C 0.000 }
gfCNCPoint1[2883] = {X 215.9094, Y 71.0067, Z -1.3333, A 0.000, B 0.000, C 0.000 }
gfCNCPoint1[2884] = {X 214.2392, Y 70.8316, Z -1.3333, A 0.000, B 0.000, C 0.000 }
gfCNCPoint1[2885] = {X 212.6095, Y 70.4266, Z -1.3333, A 0.000, B 0.000, C 0.000 }
gfCNCPoint1[2886] = {X 211.0517, Y 69.7995, Z -1.3333, A 0.000, B 0.000, C 0.000 }
gfCNCPoint1[2887] = {X 209.5959, Y 68.9624, Z -1.3333, A 0.000, B 0.000, C 0.000 }
gfCNCPoint1[2888] = {X 208.2702, Y 67.9315, Z -1.3333, A 0.000, B 0.000, C 0.000 }
gfCNCPoint1[2889] = {X 207.1004, Y 66.7267, Z -1.3333, A 0.000, B 0.000, C 0.000 }
gfCNCPoint1[2890] = {X 206.1089, Y 65.3714, Z -1.3333, A 0.000, B 0.000, C 0.000 }
gfCNCPoint1[2891] = {X 205.3149, Y 63.8916, Z -1.3333, A 0.000, B 0.000, C 0.000 }
gfCNCPoint1[2892] = {X 204.7339, Y 62.3160, Z -1.3333, A 0.000, B 0.000, C 0.000 }
gfCNCPoint1[2893] = {X 204.3769, Y 60.6751, Z -1.3333, A 0.000, B 0.000, C 0.000 }
gfCNCPoint1[2894] = {X 204.2510, Y 59.0005, Z -1.3333, A 0.000, B 0.000, C 0.000 }
gfCNCPoint1[2895] = {X 204.2508, Y 58.0000, Z -1.3333, A 0.000, B 0.000, C 0.000 }
gfCNCPoint1[2896] = {X 204.3397, Y 56.5374, Z -1.3333, A 0.000, B 0.000, C 0.000 }
gfCNCPoint1[2897] = {X 204.6050, Y 55.0963, Z -1.3333, A 0.000, B 0.000, C 0.000 }
gfCNCPoint1[2898] = {X 205.0428, Y 53.6979, Z -1.3333, A 0.000, B 0.000, C 0.000 }
gfCNCPoint1[2899] = {X 205.6468, Y 52.3629, Z -1.3333, A 0.000, B 0.000, C 0.000 }
gfCNCPoint1[2900] = {X 206.5302, Y 50.9378, Z -1.3333, A 0.000, B 0.000, C 0.000 }
gfCNCPoint1[2901] = {X 207.6025, Y 49.6488, Z -1.3333, A 0.000, B 0.000, C 0.000 }
gfCNCPoint1[2902] = {X 208.8430, Y 48.5206, Z -1.3333, A 0.000, B 0.000, C 0.000 }
gfCNCPoint1[2903] = {X 210.2277, Y 47.5751, Z -1.3333, A 0.000, B 0.000, C 0.000 }
gfCNCPoint1[2904] = {X 209.8801, Y 46.3328, Z -1.3333, A 0.000, B 0.000, C 0.000 }
gfCNCPoint1[2905] = {X 209.7572, Y 45.0487, Z -1.3333, A 0.000, B 0.000, C 0.000 }
gfCNCPoint1[2906] = {X 209.7570, Y 44.2008, Z -1.3333, A 0.000, B 0.000, C 0.000 }
gfCNCPoint1[2907] = {X 209.8559, Y 43.0097, Z -1.3333, A 0.000, B 0.000, C 0.000 }
gfCNCPoint1[2908] = {X 210.1500, Y 41.8513, Z -1.3333, A 0.000, B 0.000, C 0.000 }
gfCNCPoint1[2909] = {X 210.6312, Y 40.7572, Z -1.3333, A 0.000, B 0.000, C 0.000 }
gfCNCPoint1[2910] = {X 211.2862, Y 39.7575, Z -1.3333, A 0.000, B 0.000, C 0.000 }
gfCNCPoint1[2911] = {X 211.2862, Y 37.0796, Z -1.3333, A 0.000, B 0.000, C 0.000 }
gfCNCPoint1[2912] = {X 211.2860, Y 17.4416, Z -1.3333, A 0.000, B 0.000, C 0.000 }
gfCNCPoint1[2913] = {X 210.6370, Y 16.4476, Z -1.3333, A 0.000, B 0.000, C 0.000 }
gfCNCPoint1[2914] = {X 210.1582, Y 15.3613, Z -1.3333, A 0.000, B 0.000, C 0.000 }
gfCNCPoint1[2915] = {X 209.8623, Y 14.2116, Z -1.3333, A 0.000, B 0.000, C 0.000 }
gfCNCPoint1[2916] = {X 209.7572, Y 13.0291, Z -1.3333, A 0.000, B 0.000, C 0.000 }
gfCNCPoint1[2917] = {X 209.7570, Y 12.1868, Z -1.3333, A 0.000, B 0.000, C 0.000 }
gfCNCPoint1[2918] = {X 209.7578, Y 12.0809, Z -1.3333, A 0.000, B 0.000, C 0.000 }
gfCNCPoint1[2919] = {X 209.7601, Y 11.9750, Z -1.3333, A 0.000, B 0.000, C 0.000 }
gfCNCPoint1[2920] = {X 209.9068, Y 10.7178, Z -1.3333, A 0.000, B 0.000, C 0.000 }
gfCNCPoint1[2921] = {X 210.2689, Y 9.5051, Z -1.3333, A 0.000, B 0.000, C 0.000 }
gfCNCPoint1[2922] = {X 207.3611, Y 9.5051, Z -1.3333, A 0.000, B 0.000, C 0.000 }
gfCNCPoint1[2923] = {X 207.3611, Y 7.1051, Z -1.3333, A 0.000, B 0.000, C 0.000 }
gfCNCPoint1[2924] = {X 191.1424, Y 7.1051, Z -1.3333, A 0.000, B 0.000, C 0.000 }
gfCNCPoint1[2925] = {X 193.0992, Y 7.6487, Z -1.3333, A 0.000, B 0.000, C 0.000 }
gfCNCPoint1[2926] = {X 194.9826, Y 8.4089, Z -1.3333, A 0.000, B 0.000, C 0.000 }
gfCNCPoint1[2927] = {X 196.7685, Y 9.3761, Z -1.3333, A 0.000, B 0.000, C 0.000 }
gfCNCPoint1[2928] = {X 198.4343, Y 10.5379, Z -1.3333, A 0.000, B 0.000, C 0.000 }
gfCNCPoint1[2929] = {X 198.8564, Y 10.8884, Z -1.3333, A 0.000, B 0.000, C 0.000 }
gfCNCPoint1[2930] = {X 199.2641, Y 11.2556, Z -1.3333, A 0.000, B 0.000, C 0.000 }
gfCNCPoint1[2931] = {X 200.3490, Y 12.3983, Z -1.3333, A 0.000, B 0.000, C 0.000 }
gfCNCPoint1[2932] = {X 201.2946, Y 13.6586, Z -1.3333, A 0.000, B 0.000, C 0.000 }
gfCNCPoint1[2933] = {X 202.0882, Y 15.0198, Z -1.3333, A 0.000, B 0.000, C 0.000 }
gfCNCPoint1[2934] = {X 202.7192, Y 16.4636, Z -1.3333, A 0.000, B 0.000, C 0.000 }
gfCNCPoint1[2935] = {X 203.2129, Y 18.1834, Z -1.3333, A 0.000, B 0.000, C 0.000 }
gfCNCPoint1[2936] = {X 203.5062, Y 19.9484, Z -1.3333, A 0.000, B 0.000, C 0.000 }
gfCNCPoint1[2937] = {X 203.5953, Y 21.7354, Z -1.3333, A 0.000, B 0.000, C 0.000 }
gfCNCPoint1[2938] = {X 203.4790, Y 23.5208, Z -1.3333, A 0.000, B 0.000, C 0.000 }
gfCNCPoint1[2939] = {X 203.1588, Y 25.2811, Z -1.3333, A 0.000, B 0.000, C 0.000 }
gfCNCPoint1[2940] = {X 202.7585, Y 26.6264, Z -1.3333, A 0.000, B 0.000, C 0.000 }
gfCNCPoint1[2941] = {X 202.2070, Y 27.9171, Z -1.3333, A 0.000, B 0.000, C 0.000 }
gfCNCPoint1[2942] = {X 201.5114, Y 29.1363, Z -1.3333, A 0.000, B 0.000, C 0.000 }
gfCNCPoint1[2943] = {X 200.6810, Y 30.2678, Z -1.3333, A 0.000, B 0.000, C 0.000 }
gfCNCPoint1[2944] = {X 199.7266, Y 31.2969, Z -1.3333, A 0.000, B 0.000, C 0.000 }
gfCNCPoint1[2945] = {X 200.5664, Y 31.8695, Z -1.3333, A 0.000, B 0.000, C 0.000 }
gfCNCPoint1[2946] = {X 201.2694, Y 32.6036, Z -1.3333, A 0.000, B 0.000, C 0.000 }
gfCNCPoint1[2947] = {X 201.8050, Y 33.4673, Z -1.3333, A 0.000, B 0.000, C 0.000 }
gfCNCPoint1[2948] = {X 204.8262, Y 39.7091, Z -1.3333, A 0.000, B 0.000, C 0.000 }
gfCNCPoint1[2949] = {X 205.1508, Y 40.5847, Z -1.3333, A 0.000, B 0.000, C 0.000 }
gfCNCPoint1[2950] = {X 205.3026, Y 41.5062, Z -1.3333, A 0.000, B 0.000, C 0.000 }
gfCNCPoint1[2951] = {X 205.2761, Y 42.4397, Z -1.3333, A 0.000, B 0.000, C 0.000 }
gfCNCPoint1[2952] = {X 205.0723, Y 43.3511, Z -1.3333, A 0.000, B 0.000, C 0.000 }
gfCNCPoint1[2953] = {X 204.6986, Y 44.2070, Z -1.3333, A 0.000, B 0.000, C 0.000 }
gfCNCPoint1[2954] = {X 204.1687, Y 44.9760, Z -1.3333, A 0.000, B 0.000, C 0.000 }
gfCNCPoint1[2955] = {X 203.5020, Y 45.6299, Z -1.3333, A 0.000, B 0.000, C 0.000 }
gfCNCPoint1[2956] = {X 202.9654, Y 46.0637, Z -1.3333, A 0.000, B 0.000, C 0.000 }
gfCNCPoint1[2957] = {X 202.2133, Y 46.5635, Z -1.3333, A 0.000, B 0.000, C 0.000 }
gfCNCPoint1[2958] = {X 201.3822, Y 46.9166, Z -1.3333, A 0.000, B 0.000, C 0.000 }
gfCNCPoint1[2959] = {X 200.5004, Y 47.1112, Z -1.3333, A 0.000, B 0.000, C 0.000 }
gfCNCPoint1[2960] = {X 199.5979, Y 47.1405, Z -1.3333, A 0.000, B 0.000, C 0.000 }
gfCNCPoint1[2961] = {X 198.7053, Y 47.0036, Z -1.3333, A 0.000, B 0.000, C 0.000 }
gfCNCPoint1[2962] = {X 197.0668, Y 47.8625, Z -1.3333, A 0.000, B 0.000, C 0.000 }
gfCNCPoint1[2963] = {X 195.3763, Y 48.6136, Z -1.3333, A 0.000, B 0.000, C 0.000 }
gfCNCPoint1[2964] = {X 193.6407, Y 49.2538, Z -1.3333, A 0.000, B 0.000, C 0.000 }
gfCNCPoint1[2965] = {X 193.0856, Y 49.4466, Z -1.3333, A 0.000, B 0.000, C 0.000 }
gfCNCPoint1[2966] = {X 191.1033, Y 49.9906, Z -1.3333, A 0.000, B 0.000, C 0.000 }
gfCNCPoint1[2967] = {X 189.0809, Y 50.3586, Z -1.3333, A 0.000, B 0.000, C 0.000 }
gfCNCPoint1[2968] = {X 186.8985, Y 50.5540, Z -1.3333, A 0.000, B 0.000, C 0.000 }
gfCNCPoint1[2969] = {X 184.7074, Y 50.5444, Z -1.3333, A 0.000, B 0.000, C 0.000 }
gfCNCPoint1[2970] = {X 184.7319, Y 50.0651, Z -1.3333, A 0.000, B 0.000, C 0.000 }
gfCNCPoint1[2971] = {X 183.1137, Y 49.9246, Z -1.3333, A 0.000, B 0.000, C 0.000 }
gfCNCPoint1[2972] = {X 181.5095, Y 49.6700, Z -1.3333, A 0.000, B 0.000, C 0.000 }
gfCNCPoint1[2973] = {X 179.6143, Y 49.1962, Z -1.3333, A 0.000, B 0.000, C 0.000 }
gfCNCPoint1[2974] = {X 177.7854, Y 48.5096, Z -1.3333, A 0.000, B 0.000, C 0.000 }
gfCNCPoint1[2975] = {X 176.0467, Y 47.6190, Z -1.3333, A 0.000, B 0.000, C 0.000 }
gfCNCPoint1[2976] = {X 174.4207, Y 46.5361, Z -1.3333, A 0.000, B 0.000, C 0.000 }
gfCNCPoint1[2977] = {X 173.1808, Y 45.4895, Z -1.3333, A 0.000, B 0.000, C 0.000 }
gfCNCPoint1[2978] = {X 172.0774, Y 44.2999, Z -1.3333, A 0.000, B 0.000, C 0.000 }
gfCNCPoint1[2979] = {X 171.1269, Y 42.9848, Z -1.3333, A 0.000, B 0.000, C 0.000 }
gfCNCPoint1[2980] = {X 170.3435, Y 41.5639, Z -1.3333, A 0.000, B 0.000, C 0.000 }
gfCNCPoint1[2981] = {X 169.7387, Y 40.0582, Z -1.3333, A 0.000, B 0.000, C 0.000 }
gfCNCPoint1[2982] = {X 169.3215, Y 38.4902, Z -1.3333, A 0.000, B 0.000, C 0.000 }
gfCNCPoint1[2983] = {X 169.0983, Y 36.8831, Z -1.3333, A 0.000, B 0.000, C 0.000 }
gfCNCPoint1[2984] = {X 169.0136, Y 35.0396, Z -1.3333, A 0.000, B 0.000, C 0.000 }
gfCNCPoint1[2985] = {X 169.1604, Y 33.2001, Z -1.3333, A 0.000, B 0.000, C 0.000 }
gfCNCPoint1[2986] = {X 169.5364, Y 31.3935, Z -1.3333, A 0.000, B 0.000, C 0.000 }
gfCNCPoint1[2987] = {X 170.1356, Y 29.6481, Z -1.3333, A 0.000, B 0.000, C 0.000 }
gfCNCPoint1[2988] = {X 170.7629, Y 28.3604, Z -1.3333, A 0.000, B 0.000, C 0.000 }
gfCNCPoint1[2989] = {X 171.5530, Y 27.1656, Z -1.3333, A 0.000, B 0.000, C 0.000 }
gfCNCPoint1[2990] = {X 172.4923, Y 26.0842, Z -1.3333, A 0.000, B 0.000, C 0.000 }
gfCNCPoint1[2991] = {X 173.5648, Y 25.1347, Z -1.3333, A 0.000, B 0.000, C 0.000 }
gfCNCPoint1[2992] = {X 174.7521, Y 24.3334, Z -1.3333, A 0.000, B 0.000, C 0.000 }
gfCNCPoint1[2993] = {X 173.9917, Y 23.9231, Z -1.3333, A 0.000, B 0.000, C 0.000 }
gfCNCPoint1[2994] = {X 173.3262, Y 23.3722, Z -1.3333, A 0.000, B 0.000, C 0.000 }
gfCNCPoint1[2995] = {X 172.7811, Y 22.7018, Z -1.3333, A 0.000, B 0.000, C 0.000 }
gfCNCPoint1[2996] = {X 172.3776, Y 21.9378, Z -1.3333, A 0.000, B 0.000, C 0.000 }
gfCNCPoint1[2997] = {X 169.7664, Y 15.5423, Z -1.3333, A 0.000, B 0.000, C 0.000 }
gfCNCPoint1[2998] = {X 169.5126, Y 14.6752, Z -1.3333, A 0.000, B 0.000, C 0.000 }
gfCNCPoint1[2999] = {X 169.4412, Y 13.7745, Z -1.3333, A 0.000, B 0.000, C 0.000 }
gfCNCPoint1[3000] = {X 169.5553, Y 12.8782, Z -1.3333, A 0.000, B 0.000, C 0.000 }
gfCNCPoint1[3001] = {X 169.8501, Y 12.0242, Z -1.3333, A 0.000, B 0.000, C 0.000 }
gfCNCPoint1[3002] = {X 170.3131, Y 11.2483, Z -1.3333, A 0.000, B 0.000, C 0.000 }
gfCNCPoint1[3003] = {X 170.9248, Y 10.5834, Z -1.3333, A 0.000, B 0.000, C 0.000 }
gfCNCPoint1[3004] = {X 171.6594, Y 10.0574, Z -1.3333, A 0.000, B 0.000, C 0.000 }
gfCNCPoint1[3005] = {X 172.2916, Y 9.6970, Z -1.3333, A 0.000, B 0.000, C 0.000 }
gfCNCPoint1[3006] = {X 173.1812, Y 9.3215, Z -1.3333, A 0.000, B 0.000, C 0.000 }
gfCNCPoint1[3007] = {X 174.1313, Y 9.1491, Z -1.3333, A 0.000, B 0.000, C 0.000 }
gfCNCPoint1[3008] = {X 175.0960, Y 9.1881, Z -1.3333, A 0.000, B 0.000, C 0.000 }
gfCNCPoint1[3009] = {X 176.0291, Y 9.4366, Z -1.3333, A 0.000, B 0.000, C 0.000 }
gfCNCPoint1[3010] = {X 178.2251, Y 8.5163, Z -1.3333, A 0.000, B 0.000, C 0.000 }
gfCNCPoint1[3011] = {X 180.5019, Y 7.8197, Z -1.3333, A 0.000, B 0.000, C 0.000 }
gfCNCPoint1[3012] = {X 182.8369, Y 7.3536, Z -1.3333, A 0.000, B 0.000, C 0.000 }
gfCNCPoint1[3013] = {X 185.2067, Y 7.1227, Z -1.3333, A 0.000, B 0.000, C 0.000 }
gfCNCPoint1[3014] = {X 187.5877, Y 7.1292, Z -1.3333, A 0.000, B 0.000, C 0.000 }
gfCNCPoint1[3015] = {X 189.9562, Y 7.3733, Z -1.3333, A 0.000, B 0.000, C 0.000 }
gfCNCPoint1[3016] = {X 191.7218, Y 7.7370, Z -1.3333, A 0.000, B 0.000, C 0.000 }
gfCNCPoint1[3017] = {X 193.4408, Y 8.2799, Z -1.3333, A 0.000, B 0.000, C 0.000 }
gfCNCPoint1[3018] = {X 195.0951, Y 8.9963, Z -1.3333, A 0.000, B 0.000, C 0.000 }
gfCNCPoint1[3019] = {X 196.6672, Y 9.8786, Z -1.3333, A 0.000, B 0.000, C 0.000 }
gfCNCPoint1[3020] = {X 198.1404, Y 10.9175, Z -1.3333, A 0.000, B 0.000, C 0.000 }
gfCNCPoint1[3021] = {X 199.2067, Y 11.8672, Z -1.3333, A 0.000, B 0.000, C 0.000 }
gfCNCPoint1[3022] = {X 200.1635, Y 12.9271, Z -1.3333, A 0.000, B 0.000, C 0.000 }
gfCNCPoint1[3023] = {X 200.9995, Y 14.0847, Z -1.3333, A 0.000, B 0.000, C 0.000 }
gfCNCPoint1[3024] = {X 201.7050, Y 15.3261, Z -1.3333, A 0.000, B 0.000, C 0.000 }
gfCNCPoint1[3025] = {X 202.2714, Y 16.6369, Z -1.3333, A 0.000, B 0.000, C 0.000 }
gfCNCPoint1[3026] = {X 202.7476, Y 18.3014, Z -1.3333, A 0.000, B 0.000, C 0.000 }
gfCNCPoint1[3027] = {X 203.0301, Y 20.0095, Z -1.3333, A 0.000, B 0.000, C 0.000 }
gfCNCPoint1[3028] = {X 203.1153, Y 21.7387, Z -1.3333, A 0.000, B 0.000, C 0.000 }
gfCNCPoint1[3029] = {X 203.0021, Y 23.4663, Z -1.3333, A 0.000, B 0.000, C 0.000 }
gfCNCPoint1[3030] = {X 202.6919, Y 25.1695, Z -1.3333, A 0.000, B 0.000, C 0.000 }
gfCNCPoint1[3031] = {X 202.2573, Y 26.5985, Z -1.3333, A 0.000, B 0.000, C 0.000 }
gfCNCPoint1[3032] = {X 201.6453, Y 27.9609, Z -1.3333, A 0.000, B 0.000, C 0.000 }
gfCNCPoint1[3033] = {X 200.8656, Y 29.2349, Z -1.3333, A 0.000, B 0.000, C 0.000 }
gfCNCPoint1[3034] = {X 199.9309, Y 30.3998, Z -1.3333, A 0.000, B 0.000, C 0.000 }
gfCNCPoint1[3035] = {X 198.8561, Y 31.4370, Z -1.3333, A 0.000, B 0.000, C 0.000 }
gfCNCPoint1[3036] = {X 199.6396, Y 31.7986, Z -1.3333, A 0.000, B 0.000, C 0.000 }
gfCNCPoint1[3037] = {X 200.3374, Y 32.3063, Z -1.3333, A 0.000, B 0.000, C 0.000 }
gfCNCPoint1[3038] = {X 200.9227, Y 32.9403, Z -1.3333, A 0.000, B 0.000, C 0.000 }
gfCNCPoint1[3039] = {X 201.3730, Y 33.6764, Z -1.3333, A 0.000, B 0.000, C 0.000 }
gfCNCPoint1[3040] = {X 204.3942, Y 39.9182, Z -1.3333, A 0.000, B 0.000, C 0.000 }
gfCNCPoint1[3041] = {X 204.7207, Y 40.8441, Z -1.3333, A 0.000, B 0.000, C 0.000 }
gfCNCPoint1[3042] = {X 204.8337, Y 41.8194, Z -1.3333, A 0.000, B 0.000, C 0.000 }
gfCNCPoint1[3043] = {X 204.7276, Y 42.7955, Z -1.3333, A 0.000, B 0.000, C 0.000 }
gfCNCPoint1[3044] = {X 204.4078, Y 43.7238, Z -1.3333, A 0.000, B 0.000, C 0.000 }
gfCNCPoint1[3045] = {X 203.8900, Y 44.5580, Z -1.3333, A 0.000, B 0.000, C 0.000 }
gfCNCPoint1[3046] = {X 203.2002, Y 45.2567, Z -1.3333, A 0.000, B 0.000, C 0.000 }
gfCNCPoint1[3047] = {X 202.6636, Y 45.6905, Z -1.3333, A 0.000, B 0.000, C 0.000 }
gfCNCPoint1[3048] = {X 201.9520, Y 46.1589, Z -1.3333, A 0.000, B 0.000, C 0.000 }
gfCNCPoint1[3049] = {X 201.1637, Y 46.4819, Z -1.3333, A 0.000, B 0.000, C 0.000 }
gfCNCPoint1[3050] = {X 200.3281, Y 46.6476, Z -1.3333, A 0.000, B 0.000, C 0.000 }
gfCNCPoint1[3051] = {X 199.4762, Y 46.6498, Z -1.3333, A 0.000, B 0.000, C 0.000 }
gfCNCPoint1[3052] = {X 198.6397, Y 46.4884, Z -1.3333, A 0.000, B 0.000, C 0.000 }
gfCNCPoint1[3053] = {X 196.9749, Y 47.3735, Z -1.3333, A 0.000, B 0.000, C 0.000 }
gfCNCPoint1[3054] = {X 195.2544, Y 48.1449, Z -1.3333, A 0.000, B 0.000, C 0.000 }
gfCNCPoint1[3055] = {X 193.4862, Y 48.7993, Z -1.3333, A 0.000, B 0.000, C 0.000 }
gfCNCPoint1[3056] = {X 192.9191, Y 48.9962, Z -1.3333, A 0.000, B 0.000, C 0.000 }
gfCNCPoint1[3057] = {X 190.9171, Y 49.5408, Z -1.3333, A 0.000, B 0.000, C 0.000 }
gfCNCPoint1[3058] = {X 188.8740, Y 49.9022, Z -1.3333, A 0.000, B 0.000, C 0.000 }
gfCNCPoint1[3059] = {X 186.8067, Y 50.0774, Z -1.3333, A 0.000, B 0.000, C 0.000 }
gfCNCPoint1[3060] = {X 184.7319, Y 50.0651, Z -1.3333, A 0.000, B 0.000, C 0.000 }
gfCNCPoint1[3061] = {X 184.7074, Y 50.5444, Z -1.3333, A 0.000, B 0.000, C 0.000 }
gfCNCPoint1[3062] = {X 185.7054, Y 51.4987, Z -1.3333, A 0.000, B 0.000, C 0.000 }
gfCNCPoint1[3063] = {X 186.5575, Y 52.5854, Z -1.3333, A 0.000, B 0.000, C 0.000 }
gfCNCPoint1[3064] = {X 187.2463, Y 53.7822, Z -1.3333, A 0.000, B 0.000, C 0.000 }
gfCNCPoint1[3065] = {X 187.7795, Y 55.1342, Z -1.3333, A 0.000, B 0.000, C 0.000 }
gfCNCPoint1[3066] = {X 188.1044, Y 56.5507, Z -1.3333, A 0.000, B 0.000, C 0.000 }
gfCNCPoint1[3067] = {X 188.2135, Y 58.0000, Z -1.3333, A 0.000, B 0.000, C 0.000 }
gfCNCPoint1[3068] = {X 188.2132, Y 59.0140, Z -1.3333, A 0.000, B 0.000, C 0.000 }
gfCNCPoint1[3069] = {X 188.2026, Y 59.3933, Z -1.3333, A 0.000, B 0.000, C 0.000 }
gfCNCPoint1[3070] = {X 188.1772, Y 59.7718, Z -1.3333, A 0.000, B 0.000, C 0.000 }
gfCNCPoint1[3071] = {X 213.5207, Y 87.4310, Z -1.3333, A 0.000, B 0.000, C 0.000 }
gfCNCPoint1[3072] = {X 214.2160, Y 87.3818, Z -1.3333, A 0.000, B 0.000, C 0.000 }
gfCNCPoint1[3073] = {X 214.9117, Y 87.3403, Z -1.3333, A 0.000, B 0.000, C 0.000 }
gfCNCPoint1[3074] = {X 234.0933, Y 75.0515, Z -1.3333, A 0.000, B 0.000, C 0.000 }
gfCNCPoint1[3075] = {X 219.6585, Y 69.3864, Z -1.3333, A 0.000, B 0.000, C 0.000 }
gfCNCPoint1[3076] = {X 218.4700, Y 68.9866, Z -1.3333, A 0.000, B 0.000, C 0.000 }
gfCNCPoint1[3077] = {X 217.2434, Y 68.7261, Z -1.3333, A 0.000, B 0.000, C 0.000 }
gfCNCPoint1[3078] = {X 215.9951, Y 68.6082, Z -1.3333, A 0.000, B 0.000, C 0.000 }
gfCNCPoint1[3079] = {X 214.5246, Y 68.4441, Z -1.3333, A 0.000, B 0.000, C 0.000 }
gfCNCPoint1[3080] = {X 213.0963, Y 68.0577, Z -1.3333, A 0.000, B 0.000, C 0.000 }
gfCNCPoint1[3081] = {X 211.7436, Y 67.4582, Z -1.3333, A 0.000, B 0.000, C 0.000 }
gfCNCPoint1[3082] = {X 210.4981, Y 66.6595, Z -1.3333, A 0.000, B 0.000, C 0.000 }
gfCNCPoint1[3083] = {X 209.3888, Y 65.6803, Z -1.3333, A 0.000, B 0.000, C 0.000 }
gfCNCPoint1[3084] = {X 208.4418, Y 64.5435, Z -1.3333, A 0.000, B 0.000, C 0.000 }
gfCNCPoint1[3085] = {X 207.6790, Y 63.2756, Z -1.3333, A 0.000, B 0.000, C 0.000 }
gfCNCPoint1[3086] = {X 207.1184, Y 61.9063, Z -1.3333, A 0.000, B 0.000, C 0.000 }
gfCNCPoint1[3087] = {X 206.7730, Y 60.4676, Z -1.3333, A 0.000, B 0.000, C 0.000 }
gfCNCPoint1[3088] = {X 206.6510, Y 58.9930, Z -1.3333, A 0.000, B 0.000, C 0.000 }
gfCNCPoint1[3089] = {X 206.6508, Y 58.0000, Z -1.3333, A 0.000, B 0.000, C 0.000 }
gfCNCPoint1[3090] = {X 206.7577, Y 56.5655, Z -1.3333, A 0.000, B 0.000, C 0.000 }
gfCNCPoint1[3091] = {X 207.0760, Y 55.1628, Z -1.3333, A 0.000, B 0.000, C 0.000 }
gfCNCPoint1[3092] = {X 207.5986, Y 53.8226, Z -1.3333, A 0.000, B 0.000, C 0.000 }
gfCNCPoint1[3093] = {X 208.3140, Y 52.5747, Z -1.3333, A 0.000, B 0.000, C 0.000 }
gfCNCPoint1[3094] = {X 209.2065, Y 51.4466, Z -1.3333, A 0.000, B 0.000, C 0.000 }
gfCNCPoint1[3095] = {X 210.2563, Y 50.4632, Z -1.3333, A 0.000, B 0.000, C 0.000 }
gfCNCPoint1[3096] = {X 211.4402, Y 49.6463, Z -1.3333, A 0.000, B 0.000, C 0.000 }
gfCNCPoint1[3097] = {X 212.5893, Y 49.0723, Z -1.3333, A 0.000, B 0.000, C 0.000 }
gfCNCPoint1[3098] = {X 213.8042, Y 48.6556, Z -1.3333, A 0.000, B 0.000, C 0.000 }
gfCNCPoint1[3099] = {X 213.2578, Y 48.0874, Z -1.3333, A 0.000, B 0.000, C 0.000 }
gfCNCPoint1[3100] = {X 212.8100, Y 47.4386, Z -1.3333, A 0.000, B 0.000, C 0.000 }
gfCNCPoint1[3101] = {X 212.4725, Y 46.7262, Z -1.3333, A 0.000, B 0.000, C 0.000 }
gfCNCPoint1[3102] = {X 212.2401, Y 45.8965, Z -1.3333, A 0.000, B 0.000, C 0.000 }
gfCNCPoint1[3103] = {X 212.1572, Y 45.0389, Z -1.3333, A 0.000, B 0.000, C 0.000 }
gfCNCPoint1[3104] = {X 212.1570, Y 44.2008, Z -1.3333, A 0.000, B 0.000, C 0.000 }
gfCNCPoint1[3105] = {X 212.2385, Y 43.3184, Z -1.3333, A 0.000, B 0.000, C 0.000 }
gfCNCPoint1[3106] = {X 212.4801, Y 42.4659, Z -1.3333, A 0.000, B 0.000, C 0.000 }
gfCNCPoint1[3107] = {X 212.8737, Y 41.6720, Z -1.3333, A 0.000, B 0.000, C 0.000 }
gfCNCPoint1[3108] = {X 213.4060, Y 40.9635, Z -1.3333, A 0.000, B 0.000, C 0.000 }
gfCNCPoint1[3109] = {X 213.6835, Y 40.6575, Z -1.3333, A 0.000, B 0.000, C 0.000 }
gfCNCPoint1[3110] = {X 213.6862, Y 40.3041, Z -1.3333, A 0.000, B 0.000, C 0.000 }
gfCNCPoint1[3111] = {X 213.6862, Y 17.4645, Z -1.3333, A 0.000, B 0.000, C 0.000 }
gfCNCPoint1[3112] = {X 213.6809, Y 16.7698, Z -1.3333, A 0.000, B 0.000, C 0.000 }
gfCNCPoint1[3113] = {X 213.6806, Y 16.5204, Z -1.3333, A 0.000, B 0.000, C 0.000 }
gfCNCPoint1[3114] = {X 213.0409, Y 15.7790, Z -1.3333, A 0.000, B 0.000, C 0.000 }
gfCNCPoint1[3115] = {X 212.5622, Y 14.9248, Z -1.3333, A 0.000, B 0.000, C 0.000 }
gfCNCPoint1[3116] = {X 212.2636, Y 13.9922, Z -1.3333, A 0.000, B 0.000, C 0.000 }
gfCNCPoint1[3117] = {X 212.1572, Y 13.0188, Z -1.3333, A 0.000, B 0.000, C 0.000 }
gfCNCPoint1[3118] = {X 212.1570, Y 12.1868, Z -1.3333, A 0.000, B 0.000, C 0.000 }
gfCNCPoint1[3119] = {X 212.2436, Y 11.2718, Z -1.3333, A 0.000, B 0.000, C 0.000 }
gfCNCPoint1[3120] = {X 212.5002, Y 10.3892, Z -1.3333, A 0.000, B 0.000, C 0.000 }
gfCNCPoint1[3121] = {X 212.9449, Y 9.5281, Z -1.3333, A 0.000, B 0.000, C 0.000 }
gfCNCPoint1[3122] = {X 213.5510, Y 8.7719, Z -1.3333, A 0.000, B 0.000, C 0.000 }
gfCNCPoint1[3123] = {X 214.2946, Y 8.1503, Z -1.3333, A 0.000, B 0.000, C 0.000 }
gfCNCPoint1[3124] = {X 215.1463, Y 7.6880, Z -1.3333, A 0.000, B 0.000, C 0.000 }
gfCNCPoint1[3125] = {X 216.0727, Y 7.4030, Z -1.3333, A 0.000, B 0.000, C 0.000 }
gfCNCPoint1[3126] = {X 217.0370, Y 7.3068, Z -1.3333, A 0.000, B 0.000, C 0.000 }
gfCNCPoint1[3127] = {X 223.4805, Y 7.3068, Z -1.3333, A 0.000, B 0.000, C 0.000 }
gfCNCPoint1[3128] = {X 224.4448, Y 7.4030, Z -1.3333, A 0.000, B 0.000, C 0.000 }
gfCNCPoint1[3129] = {X 225.3712, Y 7.6880, Z -1.3333, A 0.000, B 0.000, C 0.000 }
gfCNCPoint1[3130] = {X 226.2229, Y 8.1503, Z -1.3333, A 0.000, B 0.000, C 0.000 }
gfCNCPoint1[3131] = {X 226.9665, Y 8.7719, Z -1.3333, A 0.000, B 0.000, C 0.000 }
gfCNCPoint1[3132] = {X 227.5726, Y 9.5281, Z -1.3333, A 0.000, B 0.000, C 0.000 }
gfCNCPoint1[3133] = {X 228.0173, Y 10.3892, Z -1.3333, A 0.000, B 0.000, C 0.000 }
gfCNCPoint1[3134] = {X 228.2739, Y 11.2718, Z -1.3333, A 0.000, B 0.000, C 0.000 }
gfCNCPoint1[3135] = {X 228.3605, Y 12.1868, Z -1.3333, A 0.000, B 0.000, C 0.000 }
gfCNCPoint1[3136] = {X 228.3603, Y 13.0237, Z -1.3333, A 0.000, B 0.000, C 0.000 }
gfCNCPoint1[3137] = {X 228.2528, Y 13.9975, Z -1.3333, A 0.000, B 0.000, C 0.000 }
gfCNCPoint1[3138] = {X 227.9530, Y 14.9301, Z -1.3333, A 0.000, B 0.000, C 0.000 }
gfCNCPoint1[3139] = {X 227.4730, Y 15.7841, Z -1.3333, A 0.000, B 0.000, C 0.000 }
gfCNCPoint1[3140] = {X 226.8320, Y 16.5250, Z -1.3333, A 0.000, B 0.000, C 0.000 }
gfCNCPoint1[3141] = {X 226.8329, Y 40.6626, Z -1.3333, A 0.000, B 0.000, C 0.000 }
gfCNCPoint1[3142] = {X 227.4736, Y 41.4036, Z -1.3333, A 0.000, B 0.000, C 0.000 }
gfCNCPoint1[3143] = {X 227.9534, Y 42.2575, Z -1.3333, A 0.000, B 0.000, C 0.000 }
gfCNCPoint1[3144] = {X 228.2530, Y 43.1902, Z -1.3333, A 0.000, B 0.000, C 0.000 }
gfCNCPoint1[3145] = {X 228.3603, Y 44.1638, Z -1.3333, A 0.000, B 0.000, C 0.000 }
gfCNCPoint1[3146] = {X 228.3605, Y 45.0000, Z -1.3333, A 0.000, B 0.000, C 0.000 }
gfCNCPoint1[3147] = {X 228.3507, Y 45.3090, Z -1.3333, A 0.000, B 0.000, C 0.000 }
gfCNCPoint1[3148] = {X 228.3214, Y 45.6167, Z -1.3333, A 0.000, B 0.000, C 0.000 }
gfCNCPoint1[3149] = {X 228.0910, Y 46.5992, Z -1.3333, A 0.000, B 0.000, C 0.000 }
gfCNCPoint1[3150] = {X 227.6635, Y 47.5134, Z -1.3333, A 0.000, B 0.000, C 0.000 }
gfCNCPoint1[3151] = {X 227.0571, Y 48.3200, Z -1.3333, A 0.000, B 0.000, C 0.000 }
gfCNCPoint1[3152] = {X 226.7053, Y 47.9934, Z -1.3333, A 0.000, B 0.000, C 0.000 }
gfCNCPoint1[3153] = {X 226.0261, Y 48.5889, Z -1.3333, A 0.000, B 0.000, C 0.000 }
gfCNCPoint1[3154] = {X 225.2396, Y 49.0331, Z -1.3333, A 0.000, B 0.000, C 0.000 }
gfCNCPoint1[3155] = {X 224.3790, Y 49.3073, Z -1.3333, A 0.000, B 0.000, C 0.000 }
gfCNCPoint1[3156] = {X 223.4805, Y 49.4000, Z -1.3333, A 0.000, B 0.000, C 0.000 }
gfCNCPoint1[3157] = {X 217.0370, Y 49.4000, Z -1.3333, A 0.000, B 0.000, C 0.000 }
gfCNCPoint1[3158] = {X 216.0579, Y 49.2897, Z -1.3333, A 0.000, B 0.000, C 0.000 }
gfCNCPoint1[3159] = {X 215.1279, Y 48.9643, Z -1.3333, A 0.000, B 0.000, C 0.000 }
gfCNCPoint1[3160] = {X 214.2936, Y 48.4400, Z -1.3333, A 0.000, B 0.000, C 0.000 }
gfCNCPoint1[3161] = {X 213.5969, Y 47.7433, Z -1.3333, A 0.000, B 0.000, C 0.000 }
gfCNCPoint1[3162] = {X 213.0727, Y 46.9091, Z -1.3333, A 0.000, B 0.000, C 0.000 }
gfCNCPoint1[3163] = {X 212.7473, Y 45.9791, Z -1.3333, A 0.000, B 0.000, C 0.000 }
gfCNCPoint1[3164] = {X 212.6370, Y 45.0000, Z -1.3333, A 0.000, B 0.000, C 0.000 }
gfCNCPoint1[3165] = {X 212.6370, Y 44.2008, Z -1.3333, A 0.000, B 0.000, C 0.000 }
gfCNCPoint1[3166] = {X 212.7104, Y 43.4063, Z -1.3333, A 0.000, B 0.000, C 0.000 }
gfCNCPoint1[3167] = {X 212.9279, Y 42.6386, Z -1.3333, A 0.000, B 0.000, C 0.000 }
gfCNCPoint1[3168] = {X 213.2823, Y 41.9238, Z -1.3333, A 0.000, B 0.000, C 0.000 }
gfCNCPoint1[3169] = {X 213.7616, Y 41.2859, Z -1.3333, A 0.000, B 0.000, C 0.000 }
gfCNCPoint1[3170] = {X 214.1621, Y 40.8442, Z -1.3333, A 0.000, B 0.000, C 0.000 }
gfCNCPoint1[3171] = {X 214.1662, Y 40.3060, Z -1.3333, A 0.000, B 0.000, C 0.000 }
gfCNCPoint1[3172] = {X 214.1662, Y 17.4626, Z -1.3333, A 0.000, B 0.000, C 0.000 }
gfCNCPoint1[3173] = {X 214.1609, Y 16.7692, Z -1.3333, A 0.000, B 0.000, C 0.000 }
gfCNCPoint1[3174] = {X 214.1603, Y 16.3074, Z -1.3333, A 0.000, B 0.000, C 0.000 }
gfCNCPoint1[3175] = {X 213.5174, Y 15.6185, Z -1.3333, A 0.000, B 0.000, C 0.000 }
gfCNCPoint1[3176] = {X 213.0359, Y 14.8086, Z -1.3333, A 0.000, B 0.000, C 0.000 }
gfCNCPoint1[3177] = {X 212.7379, Y 13.9147, Z -1.3333, A 0.000, B 0.000, C 0.000 }
gfCNCPoint1[3178] = {X 212.6370, Y 12.9779, Z -1.3333, A 0.000, B 0.000, C 0.000 }
gfCNCPoint1[3179] = {X 212.6370, Y 12.1868, Z -1.3333, A 0.000, B 0.000, C 0.000 }
gfCNCPoint1[3180] = {X 212.7473, Y 11.2077, Z -1.3333, A 0.000, B 0.000, C 0.000 }
gfCNCPoint1[3181] = {X 213.0728, Y 10.2777, Z -1.3333, A 0.000, B 0.000, C 0.000 }
gfCNCPoint1[3182] = {X 213.5970, Y 9.4435, Z -1.3333, A 0.000, B 0.000, C 0.000 }
gfCNCPoint1[3183] = {X 214.2937, Y 8.7468, Z -1.3333, A 0.000, B 0.000, C 0.000 }
gfCNCPoint1[3184] = {X 215.1279, Y 8.2226, Z -1.3333, A 0.000, B 0.000, C 0.000 }
gfCNCPoint1[3185] = {X 216.0579, Y 7.8971, Z -1.3333, A 0.000, B 0.000, C 0.000 }
gfCNCPoint1[3186] = {X 217.0370, Y 7.7868, Z -1.3333, A 0.000, B 0.000, C 0.000 }
gfCNCPoint1[3187] = {X 223.4805, Y 7.7868, Z -1.3333, A 0.000, B 0.000, C 0.000 }
gfCNCPoint1[3188] = {X 224.4596, Y 7.8971, Z -1.3333, A 0.000, B 0.000, C 0.000 }
gfCNCPoint1[3189] = {X 225.3896, Y 8.2226, Z -1.3333, A 0.000, B 0.000, C 0.000 }
gfCNCPoint1[3190] = {X 226.2238, Y 8.7468, Z -1.3333, A 0.000, B 0.000, C 0.000 }
gfCNCPoint1[3191] = {X 226.9205, Y 9.4435, Z -1.3333, A 0.000, B 0.000, C 0.000 }
gfCNCPoint1[3192] = {X 227.4447, Y 10.2777, Z -1.3333, A 0.000, B 0.000, C 0.000 }
gfCNCPoint1[3193] = {X 227.7702, Y 11.2077, Z -1.3333, A 0.000, B 0.000, C 0.000 }
gfCNCPoint1[3194] = {X 227.8805, Y 12.1868, Z -1.3333, A 0.000, B 0.000, C 0.000 }
gfCNCPoint1[3195] = {X 227.8802, Y 13.0233, Z -1.3333, A 0.000, B 0.000, C 0.000 }
gfCNCPoint1[3196] = {X 227.7719, Y 13.9496, Z -1.3333, A 0.000, B 0.000, C 0.000 }
gfCNCPoint1[3197] = {X 227.4707, Y 14.8323, Z -1.3333, A 0.000, B 0.000, C 0.000 }
gfCNCPoint1[3198] = {X 226.9902, Y 15.6317, Z -1.3333, A 0.000, B 0.000, C 0.000 }
gfCNCPoint1[3199] = {X 226.3520, Y 16.3118, Z -1.3333, A 0.000, B 0.000, C 0.000 }
gfCNCPoint1[3200] = {X 226.3529, Y 40.8758, Z -1.3333, A 0.000, B 0.000, C 0.000 }
gfCNCPoint1[3201] = {X 226.9976, Y 41.5649, Z -1.3333, A 0.000, B 0.000, C 0.000 }
gfCNCPoint1[3202] = {X 227.4804, Y 42.3757, Z -1.3333, A 0.000, B 0.000, C 0.000 }
gfCNCPoint1[3203] = {X 227.7793, Y 43.2707, Z -1.3333, A 0.000, B 0.000, C 0.000 }
gfCNCPoint1[3204] = {X 227.8805, Y 44.2089, Z -1.3333, A 0.000, B 0.000, C 0.000 }
gfCNCPoint1[3205] = {X 227.8805, Y 45.0000, Z -1.3333, A 0.000, B 0.000, C 0.000 }
gfCNCPoint1[3206] = {X 227.8037, Y 45.8182, Z -1.3333, A 0.000, B 0.000, C 0.000 }
gfCNCPoint1[3207] = {X 227.5762, Y 46.6079, Z -1.3333, A 0.000, B 0.000, C 0.000 }
gfCNCPoint1[3208] = {X 227.2057, Y 47.3415, Z -1.3333, A 0.000, B 0.000, C 0.000 }
gfCNCPoint1[3209] = {X 226.7053, Y 47.9934, Z -1.3333, A 0.000, B 0.000, C 0.000 }
gfCNCPoint1[3210] = {X 227.0571, Y 48.3200, Z -1.3333, A 0.000, B 0.000, C 0.000 }
gfCNCPoint1[3211] = {X 236.2309, Y 48.3200, Z -1.3333, A 0.000, B 0.000, C 0.000 }
gfCNCPoint1[3212] = {X 235.6245, Y 47.5134, Z -1.3333, A 0.000, B 0.000, C 0.000 }
gfCNCPoint1[3213] = {X 235.1970, Y 46.5992, Z -1.3333, A 0.000, B 0.000, C 0.000 }
gfCNCPoint1[3214] = {X 234.9666, Y 45.6167, Z -1.3333, A 0.000, B 0.000, C 0.000 }
gfCNCPoint1[3215] = {X 234.9373, Y 45.3090, Z -1.3333, A 0.000, B 0.000, C 0.000 }
gfCNCPoint1[3216] = {X 234.9275, Y 45.0000, Z -1.3333, A 0.000, B 0.000, C 0.000 }
gfCNCPoint1[3217] = {X 234.9275, Y 44.2089, Z -1.3333, A 0.000, B 0.000, C 0.000 }
gfCNCPoint1[3218] = {X 235.0194, Y 43.2661, Z -1.3333, A 0.000, B 0.000, C 0.000 }
gfCNCPoint1[3219] = {X 235.2917, Y 42.3588, Z -1.3333, A 0.000, B 0.000, C 0.000 }
gfCNCPoint1[3220] = {X 235.7342, Y 41.5213, Z -1.3333, A 0.000, B 0.000, C 0.000 }
gfCNCPoint1[3221] = {X 236.3302, Y 40.7849, Z -1.3333, A 0.000, B 0.000, C 0.000 }
gfCNCPoint1[3222] = {X 237.0572, Y 40.1776, Z -1.3333, A 0.000, B 0.000, C 0.000 }
gfCNCPoint1[3223] = {X 237.8878, Y 39.7222, Z -1.3333, A 0.000, B 0.000, C 0.000 }
gfCNCPoint1[3224] = {X 241.5469, Y 32.5600, Z -1.3333, A 0.000, B 0.000, C 0.000 }
gfCNCPoint1[3225] = {X 240.2126, Y 31.5575, Z -1.3333, A 0.000, B 0.000, C 0.000 }
gfCNCPoint1[3226] = {X 239.0320, Y 30.3778, Z -1.3333, A 0.000, B 0.000, C 0.000 }
gfCNCPoint1[3227] = {X 238.0285, Y 29.0442, Z -1.3333, A 0.000, B 0.000, C 0.000 }
gfCNCPoint1[3228] = {X 237.2218, Y 27.5832, Z -1.3333, A 0.000, B 0.000, C 0.000 }
gfCNCPoint1[3229] = {X 236.6279, Y 26.0235, Z -1.3333, A 0.000, B 0.000, C 0.000 }
gfCNCPoint1[3230] = {X 236.1927, Y 24.1499, Z -1.3333, A 0.000, B 0.000, C 0.000 }
gfCNCPoint1[3231] = {X 235.9708, Y 22.2393, Z -1.3333, A 0.000, B 0.000, C 0.000 }
gfCNCPoint1[3232] = {X 235.9650, Y 20.3158, Z -1.3333, A 0.000, B 0.000, C 0.000 }
gfCNCPoint1[3233] = {X 236.1752, Y 18.4039, Z -1.3333, A 0.000, B 0.000, C 0.000 }
gfCNCPoint1[3234] = {X 236.5989, Y 16.5277, Z -1.3333, A 0.000, B 0.000, C 0.000 }
gfCNCPoint1[3235] = {X 237.1181, Y 15.0571, Z -1.3333, A 0.000, B 0.000, C 0.000 }
gfCNCPoint1[3236] = {X 237.8178, Y 13.6633, Z -1.3333, A 0.000, B 0.000, C 0.000 }
gfCNCPoint1[3237] = {X 238.6868, Y 12.3683, Z -1.3333, A 0.000, B 0.000, C 0.000 }
gfCNCPoint1[3238] = {X 239.7114, Y 11.1925, Z -1.3333, A 0.000, B 0.000, C 0.000 }
gfCNCPoint1[3239] = {X 240.8755, Y 10.1546, Z -1.3333, A 0.000, B 0.000, C 0.000 }
gfCNCPoint1[3240] = {X 242.1607, Y 9.2709, Z -1.3333, A 0.000, B 0.000, C 0.000 }
gfCNCPoint1[3241] = {X 243.5466, Y 8.5555, Z -1.3333, A 0.000, B 0.000, C 0.000 }
gfCNCPoint1[3242] = {X 245.0113, Y 8.0196, Z -1.3333, A 0.000, B 0.000, C 0.000 }
gfCNCPoint1[3243] = {X 246.5316, Y 7.6718, Z -1.3333, A 0.000, B 0.000, C 0.000 }
gfCNCPoint1[3244] = {X 248.6761, Y 7.3943, Z -1.3333, A 0.000, B 0.000, C 0.000 }
gfCNCPoint1[3245] = {X 250.8369, Y 7.3119, Z -1.3333, A 0.000, B 0.000, C 0.000 }
gfCNCPoint1[3246] = {X 266.7608, Y 7.3119, Z -1.3333, A 0.000, B 0.000, C 0.000 }
gfCNCPoint1[3247] = {X 267.7189, Y 7.4133, Z -1.3333, A 0.000, B 0.000, C 0.000 }
gfCNCPoint1[3248] = {X 268.6385, Y 7.7010, Z -1.3333, A 0.000, B 0.000, C 0.000 }
gfCNCPoint1[3249] = {X 269.4837, Y 8.1635, Z -1.3333, A 0.000, B 0.000, C 0.000 }
gfCNCPoint1[3250] = {X 270.2216, Y 8.7831, Z -1.3333, A 0.000, B 0.000, C 0.000 }
gfCNCPoint1[3251] = {X 270.8235, Y 9.5355, Z -1.3333, A 0.000, B 0.000, C 0.000 }
gfCNCPoint1[3252] = {X 271.2659, Y 10.3914, Z -1.3333, A 0.000, B 0.000, C 0.000 }
gfCNCPoint1[3253] = {X 271.5231, Y 11.2720, Z -1.3333, A 0.000, B 0.000, C 0.000 }
gfCNCPoint1[3254] = {X 271.6110, Y 12.1852, Z -1.3333, A 0.000, B 0.000, C 0.000 }
gfCNCPoint1[3255] = {X 271.6108, Y 13.0282, Z -1.3333, A 0.000, B 0.000, C 0.000 }
gfCNCPoint1[3256] = {X 271.5123, Y 13.9546, Z -1.3333, A 0.000, B 0.000, C 0.000 }
gfCNCPoint1[3257] = {X 271.2396, Y 14.8453, Z -1.3333, A 0.000, B 0.000, C 0.000 }
gfCNCPoint1[3258] = {X 275.6743, Y 16.6820, Z -1.3333, A 0.000, B 0.000, C 0.000 }
gfCNCPoint1[3259] = {X 275.3121, Y 17.4576, Z -1.3333, A 0.000, B 0.000, C 0.000 }
gfCNCPoint1[3260] = {X 274.8828, Y 18.1982, Z -1.3333, A 0.000, B 0.000, C 0.000 }
gfCNCPoint1[3261] = {X 274.8827, Y 38.9883, Z -1.3333, A 0.000, B 0.000, C 0.000 }
gfCNCPoint1[3262] = {X 275.3138, Y 39.7324, Z -1.3333, A 0.000, B 0.000, C 0.000 }
gfCNCPoint1[3263] = {X 275.6773, Y 40.5119, Z -1.3333, A 0.000, B 0.000, C 0.000 }
gfCNCPoint1[3264] = {X 276.0386, Y 39.7369, Z -1.3333, A 0.000, B 0.000, C 0.000 }
gfCNCPoint1[3265] = {X 276.4665, Y 38.9967, Z -1.3333, A 0.000, B 0.000, C 0.000 }
gfCNCPoint1[3266] = {X 276.4661, Y 18.1987, Z -1.3333, A 0.000, B 0.000, C 0.000 }
gfCNCPoint1[3267] = {X 276.0367, Y 17.4579, Z -1.3333, A 0.000, B 0.000, C 0.000 }
gfCNCPoint1[3268] = {X 275.6743, Y 16.6820, Z -1.3333, A 0.000, B 0.000, C 0.000 }
gfCNCPoint1[3269] = {X 273.4570, Y 15.7637, Z -1.3333, A 0.000, B 0.000, C 0.000 }
gfCNCPoint1[3270] = {X 273.0260, Y 16.6348, Z -1.3333, A 0.000, B 0.000, C 0.000 }
gfCNCPoint1[3271] = {X 272.4828, Y 17.4407, Z -1.3333, A 0.000, B 0.000, C 0.000 }
gfCNCPoint1[3272] = {X 272.4826, Y 39.7459, Z -1.3333, A 0.000, B 0.000, C 0.000 }
gfCNCPoint1[3273] = {X 273.0274, Y 40.5544, Z -1.3333, A 0.000, B 0.000, C 0.000 }
gfCNCPoint1[3274] = {X 273.4592, Y 41.4285, Z -1.3333, A 0.000, B 0.000, C 0.000 }
gfCNCPoint1[3275] = {X 273.7591, Y 42.3102, Z -1.3333, A 0.000, B 0.000, C 0.000 }
gfCNCPoint1[3276] = {X 273.9440, Y 43.2229, Z -1.3333, A 0.000, B 0.000, C 0.000 }
gfCNCPoint1[3277] = {X 274.0108, Y 44.1519, Z -1.3333, A 0.000, B 0.000, C 0.000 }
gfCNCPoint1[3278] = {X 274.0110, Y 45.0000, Z -1.3333, A 0.000, B 0.000, C 0.000 }
gfCNCPoint1[3279] = {X 273.9884, Y 45.5734, Z -1.3333, A 0.000, B 0.000, C 0.000 }
gfCNCPoint1[3280] = {X 273.9207, Y 46.1433, Z -1.3333, A 0.000, B 0.000, C 0.000 }
gfCNCPoint1[3281] = {X 275.0713, Y 45.9760, Z -1.3333, A 0.000, B 0.000, C 0.000 }
gfCNCPoint1[3282] = {X 276.2327, Y 45.9200, Z -1.3333, A 0.000, B 0.000, C 0.000 }
gfCNCPoint1[3283] = {X 277.3960, Y 45.9200, Z -1.3333, A 0.000, B 0.000, C 0.000 }
gfCNCPoint1[3284] = {X 277.3539, Y 45.4857, Z -1.3333, A 0.000, B 0.000, C 0.000 }
gfCNCPoint1[3285] = {X 277.3378, Y 45.0497, Z -1.3333, A 0.000, B 0.000, C 0.000 }
gfCNCPoint1[3286] = {X 277.3377, Y 44.1964, Z -1.3333, A 0.000, B 0.000, C 0.000 }
gfCNCPoint1[3287] = {X 277.4035, Y 43.2526, Z -1.3333, A 0.000, B 0.000, C 0.000 }
gfCNCPoint1[3288] = {X 277.5903, Y 42.3252, Z -1.3333, A 0.000, B 0.000, C 0.000 }
gfCNCPoint1[3289] = {X 277.8949, Y 41.4295, Z -1.3333, A 0.000, B 0.000, C 0.000 }
gfCNCPoint1[3290] = {X 278.3250, Y 40.5584, Z -1.3333, A 0.000, B 0.000, C 0.000 }
gfCNCPoint1[3291] = {X 278.8665, Y 39.7517, Z -1.3333, A 0.000, B 0.000, C 0.000 }
gfCNCPoint1[3292] = {X 278.8661, Y 17.4410, Z -1.3333, A 0.000, B 0.000, C 0.000 }
gfCNCPoint1[3293] = {X 278.3228, Y 16.6349, Z -1.3333, A 0.000, B 0.000, C 0.000 }
gfCNCPoint1[3294] = {X 277.8917, Y 15.7637, Z -1.3333, A 0.000, B 0.000, C 0.000 }
gfCNCPoint1[3295] = {X 277.5902, Y 14.8788, Z -1.3333, A 0.000, B 0.000, C 0.000 }
gfCNCPoint1[3296] = {X 277.4046, Y 13.9627, Z -1.3333, A 0.000, B 0.000, C 0.000 }
gfCNCPoint1[3297] = {X 277.3379, Y 13.0303, Z -1.3333, A 0.000, B 0.000, C 0.000 }
gfCNCPoint1[3298] = {X 277.3377, Y 12.1868, Z -1.3333, A 0.000, B 0.000, C 0.000 }
gfCNCPoint1[3299] = {X 277.3952, Y 11.2738, Z -1.3333, A 0.000, B 0.000, C 0.000 }
gfCNCPoint1[3300] = {X 277.5667, Y 10.3751, Z -1.3333, A 0.000, B 0.000, C 0.000 }
gfCNCPoint1[3301] = {X 277.8496, Y 9.5051, Z -1.3333, A 0.000, B 0.000, C 0.000 }
gfCNCPoint1[3302] = {X 273.4963, Y 9.5051, Z -1.3333, A 0.000, B 0.000, C 0.000 }
gfCNCPoint1[3303] = {X 273.7796, Y 10.3730, Z -1.3333, A 0.000, B 0.000, C 0.000 }
gfCNCPoint1[3304] = {X 273.9521, Y 11.2696, Z -1.3333, A 0.000, B 0.000, C 0.000 }
gfCNCPoint1[3305] = {X 274.0110, Y 12.1806, Z -1.3333, A 0.000, B 0.000, C 0.000 }
gfCNCPoint1[3306] = {X 274.0106, Y 13.0529, Z -1.3333, A 0.000, B 0.000, C 0.000 }
gfCNCPoint1[3307] = {X 273.9421, Y 13.9776, Z -1.3333, A 0.000, B 0.000, C 0.000 }
gfCNCPoint1[3308] = {X 273.7565, Y 14.8861, Z -1.3333, A 0.000, B 0.000, C 0.000 }
gfCNCPoint1[3309] = {X 273.4570, Y 15.7637, Z -1.3333, A 0.000, B 0.000, C 0.000 }
gfCNCPoint1[3310] = {X 271.2396, Y 14.8453, Z -1.3333, A 0.000, B 0.000, C 0.000 }
gfCNCPoint1[3311] = {X 270.7500, Y 15.7462, Z -1.3333, A 0.000, B 0.000, C 0.000 }
gfCNCPoint1[3312] = {X 270.0828, Y 16.5248, Z -1.3333, A 0.000, B 0.000, C 0.000 }
gfCNCPoint1[3313] = {X 270.0826, Y 40.6618, Z -1.3333, A 0.000, B 0.000, C 0.000 }
gfCNCPoint1[3314] = {X 270.7236, Y 41.4028, Z -1.3333, A 0.000, B 0.000, C 0.000 }
gfCNCPoint1[3315] = {X 271.2036, Y 42.2568, Z -1.3333, A 0.000, B 0.000, C 0.000 }
gfCNCPoint1[3316] = {X 271.5034, Y 43.1895, Z -1.3333, A 0.000, B 0.000, C 0.000 }
gfCNCPoint1[3317] = {X 271.6108, Y 44.1633, Z -1.3333, A 0.000, B 0.000, C 0.000 }
gfCNCPoint1[3318] = {X 271.6110, Y 45.0000, Z -1.3333, A 0.000, B 0.000, C 0.000 }
gfCNCPoint1[3319] = {X 271.5959, Y 45.3844, Z -1.3333, A 0.000, B 0.000, C 0.000 }
gfCNCPoint1[3320] = {X 271.5505, Y 45.7664, Z -1.3333, A 0.000, B 0.000, C 0.000 }
gfCNCPoint1[3321] = {X 271.2989, Y 46.7171, Z -1.3333, A 0.000, B 0.000, C 0.000 }
gfCNCPoint1[3322] = {X 270.8619, Y 47.5982, Z -1.3333, A 0.000, B 0.000, C 0.000 }
gfCNCPoint1[3323] = {X 270.2571, Y 48.3736, Z -1.3333, A 0.000, B 0.000, C 0.000 }
gfCNCPoint1[3324] = {X 269.5090, Y 49.0121, Z -1.3333, A 0.000, B 0.000, C 0.000 }
gfCNCPoint1[3325] = {X 268.6482, Y 49.4876, Z -1.3333, A 0.000, B 0.000, C 0.000 }
gfCNCPoint1[3326] = {X 267.7095, Y 49.7809, Z -1.3333, A 0.000, B 0.000, C 0.000 }
gfCNCPoint1[3327] = {X 266.7310, Y 49.8800, Z -1.3333, A 0.000, B 0.000, C 0.000 }
gfCNCPoint1[3328] = {X 260.2876, Y 49.8800, Z -1.3333, A 0.000, B 0.000, C 0.000 }
gfCNCPoint1[3329] = {X 259.3713, Y 49.7932, Z -1.3333, A 0.000, B 0.000, C 0.000 }
gfCNCPoint1[3330] = {X 258.4877, Y 49.5359, Z -1.3333, A 0.000, B 0.000, C 0.000 }
gfCNCPoint1[3331] = {X 257.6680, Y 49.1173, Z -1.3333, A 0.000, B 0.000, C 0.000 }
gfCNCPoint1[3332] = {X 256.9416, Y 48.5523, Z -1.3333, A 0.000, B 0.000, C 0.000 }
gfCNCPoint1[3333] = {X 253.6505, Y 52.0464, Z -1.3333, A 0.000, B 0.000, C 0.000 }
gfCNCPoint1[3334] = {X 253.4938, Y 51.8954, Z -1.3333, A 0.000, B 0.000, C 0.000 }
gfCNCPoint1[3335] = {X 253.3406, Y 51.7410, Z -1.3333, A 0.000, B 0.000, C 0.000 }
gfCNCPoint1[3336] = {X 253.2761, Y 51.8068, Z -1.3333, A 0.000, B 0.000, C 0.000 }
gfCNCPoint1[3337] = {X 253.2111, Y 51.8720, Z -1.3333, A 0.000, B 0.000, C 0.000 }
gfCNCPoint1[3338] = {X 253.6505, Y 52.0464, Z -1.3333, A 0.000, B 0.000, C 0.000 }
gfCNCPoint1[3339] = {X 255.2960, Y 50.2993, Z -1.3333, A 0.000, B 0.000, C 0.000 }
gfCNCPoint1[3340] = {X 255.1782, Y 50.1858, Z -1.3333, A 0.000, B 0.000, C 0.000 }
gfCNCPoint1[3341] = {X 255.0630, Y 50.0697, Z -1.3333, A 0.000, B 0.000, C 0.000 }
gfCNCPoint1[3342] = {X 254.3405, Y 49.1989, Z -1.3333, A 0.000, B 0.000, C 0.000 }
gfCNCPoint1[3343] = {X 253.7617, Y 48.2267, Z -1.3333, A 0.000, B 0.000, C 0.000 }
gfCNCPoint1[3344] = {X 253.3406, Y 47.1766, Z -1.3333, A 0.000, B 0.000, C 0.000 }
gfCNCPoint1[3345] = {X 252.9194, Y 48.2267, Z -1.3333, A 0.000, B 0.000, C 0.000 }
gfCNCPoint1[3346] = {X 252.3406, Y 49.1989, Z -1.3333, A 0.000, B 0.000, C 0.000 }
gfCNCPoint1[3347] = {X 251.6182, Y 50.0697, Z -1.3333, A 0.000, B 0.000, C 0.000 }
gfCNCPoint1[3348] = {X 251.5697, Y 50.1192, Z -1.3333, A 0.000, B 0.000, C 0.000 }
gfCNCPoint1[3349] = {X 251.5208, Y 50.1682, Z -1.3333, A 0.000, B 0.000, C 0.000 }
gfCNCPoint1[3350] = {X 250.7149, Y 50.8587, Z -1.3333, A 0.000, B 0.000, C 0.000 }
gfCNCPoint1[3351] = {X 249.8172, Y 51.4247, Z -1.3333, A 0.000, B 0.000, C 0.000 }
gfCNCPoint1[3352] = {X 248.8467, Y 51.8542, Z -1.3333, A 0.000, B 0.000, C 0.000 }
gfCNCPoint1[3353] = {X 247.8241, Y 52.1381, Z -1.3333, A 0.000, B 0.000, C 0.000 }
gfCNCPoint1[3354] = {X 247.8931, Y 52.2642, Z -1.3333, A 0.000, B 0.000, C 0.000 }
gfCNCPoint1[3355] = {X 247.9606, Y 52.3912, Z -1.3333, A 0.000, B 0.000, C 0.000 }
gfCNCPoint1[3356] = {X 250.9656, Y 53.5628, Z -1.3333, A 0.000, B 0.000, C 0.000 }
gfCNCPoint1[3357] = {X 259.4003, Y 56.9107, Z -1.3333, A 0.000, B 0.000, C 0.000 }
gfCNCPoint1[3358] = {X 260.2857, Y 54.6800, Z -1.3333, A 0.000, B 0.000, C 0.000 }
gfCNCPoint1[3359] = {X 261.9956, Y 55.3587, Z -1.3333, A 0.000, B 0.000, C 0.000 }
gfCNCPoint1[3360] = {X 262.0630, Y 55.0185, Z -1.3333, A 0.000, B 0.000, C 0.000 }
gfCNCPoint1[3361] = {X 262.1384, Y 54.6800, Z -1.3333, A 0.000, B 0.000, C 0.000 }
gfCNCPoint1[3362] = {X 260.2857, Y 54.6800, Z -1.3333, A 0.000, B 0.000, C 0.000 }
gfCNCPoint1[3363] = {X 259.4003, Y 56.9107, Z -1.3333, A 0.000, B 0.000, C 0.000 }
gfCNCPoint1[3364] = {X 264.1528, Y 58.7971, Z -1.3333, A 0.000, B 0.000, C 0.000 }
gfCNCPoint1[3365] = {X 264.1527, Y 58.0000, Z -1.3333, A 0.000, B 0.000, C 0.000 }
gfCNCPoint1[3366] = {X 264.2035, Y 56.8936, Z -1.3333, A 0.000, B 0.000, C 0.000 }
gfCNCPoint1[3367] = {X 264.3554, Y 55.7965, Z -1.3333, A 0.000, B 0.000, C 0.000 }
gfCNCPoint1[3368] = {X 264.4115, Y 55.5127, Z -1.3333, A 0.000, B 0.000, C 0.000 }
gfCNCPoint1[3369] = {X 264.4745, Y 55.2303, Z -1.3333, A 0.000, B 0.000, C 0.000 }
gfCNCPoint1[3370] = {X 264.9369, Y 53.7185, Z -1.3333, A 0.000, B 0.000, C 0.000 }
gfCNCPoint1[3371] = {X 265.5928, Y 52.2800, Z -1.3333, A 0.000, B 0.000, C 0.000 }
gfCNCPoint1[3372] = {X 260.2876, Y 52.2800, Z -1.3333, A 0.000, B 0.000, C 0.000 }
gfCNCPoint1[3373] = {X 259.1917, Y 52.1971, Z -1.3333, A 0.000, B 0.000, C 0.000 }
gfCNCPoint1[3374] = {X 258.1209, Y 51.9501, Z -1.3333, A 0.000, B 0.000, C 0.000 }
gfCNCPoint1[3375] = {X 257.0994, Y 51.5448, Z -1.3333, A 0.000, B 0.000, C 0.000 }
gfCNCPoint1[3376] = {X 256.1506, Y 50.9903, Z -1.3333, A 0.000, B 0.000, C 0.000 }
gfCNCPoint1[3377] = {X 255.2960, Y 50.2993, Z -1.3333, A 0.000, B 0.000, C 0.000 }
gfCNCPoint1[3378] = {X 256.9416, Y 48.5523, Z -1.3333, A 0.000, B 0.000, C 0.000 }
gfCNCPoint1[3379] = {X 256.3872, Y 47.9328, Z -1.3333, A 0.000, B 0.000, C 0.000 }
gfCNCPoint1[3380] = {X 255.9460, Y 47.2283, Z -1.3333, A 0.000, B 0.000, C 0.000 }
gfCNCPoint1[3381] = {X 255.6308, Y 46.4590, Z -1.3333, A 0.000, B 0.000, C 0.000 }
gfCNCPoint1[3382] = {X 255.4666, Y 45.7568, Z -1.3333, A 0.000, B 0.000, C 0.000 }
gfCNCPoint1[3383] = {X 255.4077, Y 45.0380, Z -1.3333, A 0.000, B 0.000, C 0.000 }
gfCNCPoint1[3384] = {X 255.4080, Y 44.1417, Z -1.3333, A 0.000, B 0.000, C 0.000 }
gfCNCPoint1[3385] = {X 255.5183, Y 43.1751, Z -1.3333, A 0.000, B 0.000, C 0.000 }
gfCNCPoint1[3386] = {X 255.8181, Y 42.2497, Z -1.3333, A 0.000, B 0.000, C 0.000 }
gfCNCPoint1[3387] = {X 256.2955, Y 41.4021, Z -1.3333, A 0.000, B 0.000, C 0.000 }
gfCNCPoint1[3388] = {X 256.9315, Y 40.6660, Z -1.3333, A 0.000, B 0.000, C 0.000 }
gfCNCPoint1[3389] = {X 256.9315, Y 35.0338, Z -1.3333, A 0.000, B 0.000, C 0.000 }
gfCNCPoint1[3390] = {X 255.1085, Y 35.0338, Z -1.3333, A 0.000, B 0.000, C 0.000 }
gfCNCPoint1[3391] = {X 251.0863, Y 42.8698, Z -1.3333, A 0.000, B 0.000, C 0.000 }
gfCNCPoint1[3392] = {X 251.2236, Y 43.5124, Z -1.3333, A 0.000, B 0.000, C 0.000 }
gfCNCPoint1[3393] = {X 251.2734, Y 44.1675, Z -1.3333, A 0.000, B 0.000, C 0.000 }
gfCNCPoint1[3394] = {X 251.2736, Y 45.0000, Z -1.3333, A 0.000, B 0.000, C 0.000 }
gfCNCPoint1[3395] = {X 251.2174, Y 45.7380, Z -1.3333, A 0.000, B 0.000, C 0.000 }
gfCNCPoint1[3396] = {X 251.0503, Y 46.4590, Z -1.3333, A 0.000, B 0.000, C 0.000 }
gfCNCPoint1[3397] = {X 250.6346, Y 47.4142, Z -1.3333, A 0.000, B 0.000, C 0.000 }
gfCNCPoint1[3398] = {X 250.0255, Y 48.2593, Z -1.3333, A 0.000, B 0.000, C 0.000 }
gfCNCPoint1[3399] = {X 249.2510, Y 48.9560, Z -1.3333, A 0.000, B 0.000, C 0.000 }
gfCNCPoint1[3400] = {X 248.3462, Y 49.4723, Z -1.3333, A 0.000, B 0.000, C 0.000 }
gfCNCPoint1[3401] = {X 247.3525, Y 49.7849, Z -1.3333, A 0.000, B 0.000, C 0.000 }
gfCNCPoint1[3402] = {X 246.8754, Y 49.8562, Z -1.3333, A 0.000, B 0.000, C 0.000 }
gfCNCPoint1[3403] = {X 246.3936, Y 49.8800, Z -1.3333, A 0.000, B 0.000, C 0.000 }
gfCNCPoint1[3404] = {X 242.5312, Y 49.8800, Z -1.3333, A 0.000, B 0.000, C 0.000 }
gfCNCPoint1[3405] = {X 242.5312, Y 49.4000, Z -1.3333, A 0.000, B 0.000, C 0.000 }
gfCNCPoint1[3406] = {X 239.8075, Y 49.4000, Z -1.3333, A 0.000, B 0.000, C 0.000 }
gfCNCPoint1[3407] = {X 238.8284, Y 49.2897, Z -1.3333, A 0.000, B 0.000, C 0.000 }
gfCNCPoint1[3408] = {X 237.8984, Y 48.9643, Z -1.3333, A 0.000, B 0.000, C 0.000 }
gfCNCPoint1[3409] = {X 237.0641, Y 48.4401, Z -1.3333, A 0.000, B 0.000, C 0.000 }
gfCNCPoint1[3410] = {X 236.3674, Y 47.7434, Z -1.3333, A 0.000, B 0.000, C 0.000 }
gfCNCPoint1[3411] = {X 235.8432, Y 46.9091, Z -1.3333, A 0.000, B 0.000, C 0.000 }
gfCNCPoint1[3412] = {X 235.5178, Y 45.9791, Z -1.3333, A 0.000, B 0.000, C 0.000 }
gfCNCPoint1[3413] = {X 235.4075, Y 45.0000, Z -1.3333, A 0.000, B 0.000, C 0.000 }
gfCNCPoint1[3414] = {X 235.4079, Y 44.1483, Z -1.3333, A 0.000, B 0.000, C 0.000 }
gfCNCPoint1[3415] = {X 235.5063, Y 43.2816, Z -1.3333, A 0.000, B 0.000, C 0.000 }
gfCNCPoint1[3416] = {X 235.7737, Y 42.4514, Z -1.3333, A 0.000, B 0.000, C 0.000 }
gfCNCPoint1[3417] = {X 236.1996, Y 41.6903, Z -1.3333, A 0.000, B 0.000, C 0.000 }
gfCNCPoint1[3418] = {X 236.7672, Y 41.0281, Z -1.3333, A 0.000, B 0.000, C 0.000 }
gfCNCPoint1[3419] = {X 237.4544, Y 40.4909, Z -1.3333, A 0.000, B 0.000, C 0.000 }
gfCNCPoint1[3420] = {X 238.2339, Y 40.0998, Z -1.3333, A 0.000, B 0.000, C 0.000 }
gfCNCPoint1[3421] = {X 242.1753, Y 32.3850, Z -1.3333, A 0.000, B 0.000, C 0.000 }
gfCNCPoint1[3422] = {X 241.0119, Y 31.5927, Z -1.3333, A 0.000, B 0.000, C 0.000 }
gfCNCPoint1[3423] = {X 239.9551, Y 30.6631, Z -1.3333, A 0.000, B 0.000, C 0.000 }
gfCNCPoint1[3424] = {X 239.0209, Y 29.6102, Z -1.3333, A 0.000, B 0.000, C 0.000 }
gfCNCPoint1[3425] = {X 238.2236, Y 28.4502, Z -1.3333, A 0.000, B 0.000, C 0.000 }
gfCNCPoint1[3426] = {X 237.5755, Y 27.2008, Z -1.3333, A 0.000, B 0.000, C 0.000 }
gfCNCPoint1[3427] = {X 237.0863, Y 25.8809, Z -1.3333, A 0.000, B 0.000, C 0.000 }
gfCNCPoint1[3428] = {X 236.6645, Y 24.0613, Z -1.3333, A 0.000, B 0.000, C 0.000 }
gfCNCPoint1[3429] = {X 236.4497, Y 22.2058, Z -1.3333, A 0.000, B 0.000, C 0.000 }
gfCNCPoint1[3430] = {X 236.4445, Y 20.3379, Z -1.3333, A 0.000, B 0.000, C 0.000 }
gfCNCPoint1[3431] = {X 236.6489, Y 18.4812, Z -1.3333, A 0.000, B 0.000, C 0.000 }
gfCNCPoint1[3432] = {X 237.0605, Y 16.6592, Z -1.3333, A 0.000, B 0.000, C 0.000 }
gfCNCPoint1[3433] = {X 237.6346, Y 15.0731, Z -1.3333, A 0.000, B 0.000, C 0.000 }
gfCNCPoint1[3434] = {X 238.4266, Y 13.5839, Z -1.3333, A 0.000, B 0.000, C 0.000 }
gfCNCPoint1[3435] = {X 239.4210, Y 12.2213, Z -1.3333, A 0.000, B 0.000, C 0.000 }
gfCNCPoint1[3436] = {X 240.5976, Y 11.0126, Z -1.3333, A 0.000, B 0.000, C 0.000 }
gfCNCPoint1[3437] = {X 241.9329, Y 9.9821, Z -1.3333, A 0.000, B 0.000, C 0.000 }
gfCNCPoint1[3438] = {X 243.4004, Y 9.1502, Z -1.3333, A 0.000, B 0.000, C 0.000 }
gfCNCPoint1[3439] = {X 244.9705, Y 8.5338, Z -1.3333, A 0.000, B 0.000, C 0.000 }
gfCNCPoint1[3440] = {X 246.6119, Y 8.1450, Z -1.3333, A 0.000, B 0.000, C 0.000 }
gfCNCPoint1[3441] = {X 248.7155, Y 7.8727, Z -1.3333, A 0.000, B 0.000, C 0.000 }
gfCNCPoint1[3442] = {X 250.8351, Y 7.7919, Z -1.3333, A 0.000, B 0.000, C 0.000 }
gfCNCPoint1[3443] = {X 266.7640, Y 7.7919, Z -1.3333, A 0.000, B 0.000, C 0.000 }
gfCNCPoint1[3444] = {X 267.7367, Y 7.9088, Z -1.3333, A 0.000, B 0.000, C 0.000 }
gfCNCPoint1[3445] = {X 268.6594, Y 8.2379, Z -1.3333, A 0.000, B 0.000, C 0.000 }
gfCNCPoint1[3446] = {X 269.4865, Y 8.7628, Z -1.3333, A 0.000, B 0.000, C 0.000 }
gfCNCPoint1[3447] = {X 270.1770, Y 9.4577, Z -1.3333, A 0.000, B 0.000, C 0.000 }
gfCNCPoint1[3448] = {X 270.6969, Y 10.2880, Z -1.3333, A 0.000, B 0.000, C 0.000 }
gfCNCPoint1[3449] = {X 271.0202, Y 11.2128, Z -1.3333, A 0.000, B 0.000, C 0.000 }
gfCNCPoint1[3450] = {X 271.1310, Y 12.1861, Z -1.3333, A 0.000, B 0.000, C 0.000 }
gfCNCPoint1[3451] = {X 271.1308, Y 13.0233, Z -1.3333, A 0.000, B 0.000, C 0.000 }
gfCNCPoint1[3452] = {X 271.0224, Y 13.9496, Z -1.3333, A 0.000, B 0.000, C 0.000 }
gfCNCPoint1[3453] = {X 270.7213, Y 14.8322, Z -1.3333, A 0.000, B 0.000, C 0.000 }
gfCNCPoint1[3454] = {X 270.2409, Y 15.6315, Z -1.3333, A 0.000, B 0.000, C 0.000 }
gfCNCPoint1[3455] = {X 269.6028, Y 16.3116, Z -1.3333, A 0.000, B 0.000, C 0.000 }
gfCNCPoint1[3456] = {X 269.6026, Y 40.8750, Z -1.3333, A 0.000, B 0.000, C 0.000 }
gfCNCPoint1[3457] = {X 270.2476, Y 41.5642, Z -1.3333, A 0.000, B 0.000, C 0.000 }
gfCNCPoint1[3458] = {X 270.7308, Y 42.3752, Z -1.3333, A 0.000, B 0.000, C 0.000 }
gfCNCPoint1[3459] = {X 271.0298, Y 43.2705, Z -1.3333, A 0.000, B 0.000, C 0.000 }
gfCNCPoint1[3460] = {X 271.1310, Y 44.2089, Z -1.3333, A 0.000, B 0.000, C 0.000 }
gfCNCPoint1[3461] = {X 271.1310, Y 45.0000, Z -1.3333, A 0.000, B 0.000, C 0.000 }
gfCNCPoint1[3462] = {X 271.0207, Y 45.9791, Z -1.3333, A 0.000, B 0.000, C 0.000 }
gfCNCPoint1[3463] = {X 270.6953, Y 46.9091, Z -1.3333, A 0.000, B 0.000, C 0.000 }
gfCNCPoint1[3464] = {X 270.1711, Y 47.7434, Z -1.3333, A 0.000, B 0.000, C 0.000 }
gfCNCPoint1[3465] = {X 269.4744, Y 48.4401, Z -1.3333, A 0.000, B 0.000, C 0.000 }
gfCNCPoint1[3466] = {X 268.6401, Y 48.9643, Z -1.3333, A 0.000, B 0.000, C 0.000 }
gfCNCPoint1[3467] = {X 267.7101, Y 49.2897, Z -1.3333, A 0.000, B 0.000, C 0.000 }
gfCNCPoint1[3468] = {X 266.7310, Y 49.4000, Z -1.3333, A 0.000, B 0.000, C 0.000 }
gfCNCPoint1[3469] = {X 260.2876, Y 49.4000, Z -1.3333, A 0.000, B 0.000, C 0.000 }
gfCNCPoint1[3470] = {X 259.3085, Y 49.2897, Z -1.3333, A 0.000, B 0.000, C 0.000 }
gfCNCPoint1[3471] = {X 258.3785, Y 48.9643, Z -1.3333, A 0.000, B 0.000, C 0.000 }
gfCNCPoint1[3472] = {X 257.5442, Y 48.4400, Z -1.3333, A 0.000, B 0.000, C 0.000 }
gfCNCPoint1[3473] = {X 256.8475, Y 47.7433, Z -1.3333, A 0.000, B 0.000, C 0.000 }
gfCNCPoint1[3474] = {X 256.3233, Y 46.9091, Z -1.3333, A 0.000, B 0.000, C 0.000 }
gfCNCPoint1[3475] = {X 255.9979, Y 45.9791, Z -1.3333, A 0.000, B 0.000, C 0.000 }
gfCNCPoint1[3476] = {X 255.8876, Y 45.0000, Z -1.3333, A 0.000, B 0.000, C 0.000 }
gfCNCPoint1[3477] = {X 255.8880, Y 44.1483, Z -1.3333, A 0.000, B 0.000, C 0.000 }
gfCNCPoint1[3478] = {X 255.9984, Y 43.2275, Z -1.3333, A 0.000, B 0.000, C 0.000 }
gfCNCPoint1[3479] = {X 256.2993, Y 42.3503, Z -1.3333, A 0.000, B 0.000, C 0.000 }
gfCNCPoint1[3480] = {X 256.7775, Y 41.5556, Z -1.3333, A 0.000, B 0.000, C 0.000 }
gfCNCPoint1[3481] = {X 257.4115, Y 40.8789, Z -1.3333, A 0.000, B 0.000, C 0.000 }
gfCNCPoint1[3482] = {X 257.4115, Y 34.5538, Z -1.3333, A 0.000, B 0.000, C 0.000 }
gfCNCPoint1[3483] = {X 254.8153, Y 34.5538, Z -1.3333, A 0.000, B 0.000, C 0.000 }
gfCNCPoint1[3484] = {X 250.5701, Y 42.8244, Z -1.3333, A 0.000, B 0.000, C 0.000 }
gfCNCPoint1[3485] = {X 250.7373, Y 43.5077, Z -1.3333, A 0.000, B 0.000, C 0.000 }
gfCNCPoint1[3486] = {X 250.7936, Y 44.2089, Z -1.3333, A 0.000, B 0.000, C 0.000 }
gfCNCPoint1[3487] = {X 250.7936, Y 45.0000, Z -1.3333, A 0.000, B 0.000, C 0.000 }
gfCNCPoint1[3488] = {X 250.6832, Y 45.9791, Z -1.3333, A 0.000, B 0.000, C 0.000 }
gfCNCPoint1[3489] = {X 250.3578, Y 46.9091, Z -1.3333, A 0.000, B 0.000, C 0.000 }
gfCNCPoint1[3490] = {X 249.8336, Y 47.7434, Z -1.3333, A 0.000, B 0.000, C 0.000 }
gfCNCPoint1[3491] = {X 249.1369, Y 48.4401, Z -1.3333, A 0.000, B 0.000, C 0.000 }
gfCNCPoint1[3492] = {X 248.3026, Y 48.9643, Z -1.3333, A 0.000, B 0.000, C 0.000 }
gfCNCPoint1[3493] = {X 247.3727, Y 49.2897, Z -1.3333, A 0.000, B 0.000, C 0.000 }
gfCNCPoint1[3494] = {X 246.3936, Y 49.4000, Z -1.3333, A 0.000, B 0.000, C 0.000 }
gfCNCPoint1[3495] = {X 242.5312, Y 49.4000, Z -1.3333, A 0.000, B 0.000, C 0.000 }
gfCNCPoint1[3496] = {X 242.5312, Y 49.8800, Z -1.3333, A 0.000, B 0.000, C 0.000 }
gfCNCPoint1[3497] = {X 243.4812, Y 50.5824, Z -1.3333, A 0.000, B 0.000, C 0.000 }
gfCNCPoint1[3498] = {X 244.3384, Y 51.3953, Z -1.3333, A 0.000, B 0.000, C 0.000 }
gfCNCPoint1[3499] = {X 245.0903, Y 52.3066, Z -1.3333, A 0.000, B 0.000, C 0.000 }
gfCNCPoint1[3500] = {X 245.7256, Y 53.3027, Z -1.3333, A 0.000, B 0.000, C 0.000 }
gfCNCPoint1[3501] = {X 245.9757, Y 53.7847, Z -1.3333, A 0.000, B 0.000, C 0.000 }
gfCNCPoint1[3502] = {X 246.1984, Y 54.2800, Z -1.3333, A 0.000, B 0.000, C 0.000 }
gfCNCPoint1[3503] = {X 250.0837, Y 55.7949, Z -1.3333, A 0.000, B 0.000, C 0.000 }
gfCNCPoint1[3504] = {X 267.2825, Y 62.6215, Z -1.3333, A 0.000, B 0.000, C 0.000 }
gfCNCPoint1[3505] = {X 266.8844, Y 61.4466, Z -1.3333, A 0.000, B 0.000, C 0.000 }
gfCNCPoint1[3506] = {X 266.6399, Y 60.2304, Z -1.3333, A 0.000, B 0.000, C 0.000 }
gfCNCPoint1[3507] = {X 266.5529, Y 58.9930, Z -1.3333, A 0.000, B 0.000, C 0.000 }
gfCNCPoint1[3508] = {X 266.5527, Y 58.0000, Z -1.3333, A 0.000, B 0.000, C 0.000 }
gfCNCPoint1[3509] = {X 266.6262, Y 56.8093, Z -1.3333, A 0.000, B 0.000, C 0.000 }
gfCNCPoint1[3510] = {X 266.8456, Y 55.6367, Z -1.3333, A 0.000, B 0.000, C 0.000 }
gfCNCPoint1[3511] = {X 267.2076, Y 54.5000, Z -1.3333, A 0.000, B 0.000, C 0.000 }
gfCNCPoint1[3512] = {X 267.7067, Y 53.4164, Z -1.3333, A 0.000, B 0.000, C 0.000 }
gfCNCPoint1[3513] = {X 268.4728, Y 52.2132, Z -1.3333, A 0.000, B 0.000, C 0.000 }
gfCNCPoint1[3514] = {X 269.4075, Y 51.1357, Z -1.3333, A 0.000, B 0.000, C 0.000 }
gfCNCPoint1[3515] = {X 270.4903, Y 50.2072, Z -1.3333, A 0.000, B 0.000, C 0.000 }
gfCNCPoint1[3516] = {X 271.6979, Y 49.4479, Z -1.3333, A 0.000, B 0.000, C 0.000 }
gfCNCPoint1[3517] = {X 273.0039, Y 48.8744, Z -1.3333, A 0.000, B 0.000, C 0.000 }
gfCNCPoint1[3518] = {X 274.3800, Y 48.4989, Z -1.3333, A 0.000, B 0.000, C 0.000 }
gfCNCPoint1[3519] = {X 275.3020, Y 48.3648, Z -1.3333, A 0.000, B 0.000, C 0.000 }
gfCNCPoint1[3520] = {X 276.2327, Y 48.3200, Z -1.3333, A 0.000, B 0.000, C 0.000 }
gfCNCPoint1[3521] = {X 281.0411, Y 48.3200, Z -1.3333, A 0.000, B 0.000, C 0.000 }
gfCNCPoint1[3522] = {X 280.4347, Y 47.5134, Z -1.3333, A 0.000, B 0.000, C 0.000 }
gfCNCPoint1[3523] = {X 280.0072, Y 46.5992, Z -1.3333, A 0.000, B 0.000, C 0.000 }
gfCNCPoint1[3524] = {X 279.7768, Y 45.6167, Z -1.3333, A 0.000, B 0.000, C 0.000 }
gfCNCPoint1[3525] = {X 279.7488, Y 45.3288, Z -1.3333, A 0.000, B 0.000, C 0.000 }
gfCNCPoint1[3526] = {X 279.7378, Y 45.0398, Z -1.3333, A 0.000, B 0.000, C 0.000 }
gfCNCPoint1[3527] = {X 279.7377, Y 44.2035, Z -1.3333, A 0.000, B 0.000, C 0.000 }
gfCNCPoint1[3528] = {X 279.8428, Y 43.2203, Z -1.3333, A 0.000, B 0.000, C 0.000 }
gfCNCPoint1[3529] = {X 280.1419, Y 42.2777, Z -1.3333, A 0.000, B 0.000, C 0.000 }
gfCNCPoint1[3530] = {X 280.6229, Y 41.4138, Z -1.3333, A 0.000, B 0.000, C 0.000 }
gfCNCPoint1[3531] = {X 281.2665, Y 40.6631, Z -1.3333, A 0.000, B 0.000, C 0.000 }
gfCNCPoint1[3532] = {X 281.2661, Y 16.5251, Z -1.3333, A 0.000, B 0.000, C 0.000 }
gfCNCPoint1[3533] = {X 280.6246, Y 15.7833, Z -1.3333, A 0.000, B 0.000, C 0.000 }
gfCNCPoint1[3534] = {X 280.1443, Y 14.9283, Z -1.3333, A 0.000, B 0.000, C 0.000 }
gfCNCPoint1[3535] = {X 279.8447, Y 13.9946, Z -1.3333, A 0.000, B 0.000, C 0.000 }
gfCNCPoint1[3536] = {X 279.7378, Y 13.0198, Z -1.3333, A 0.000, B 0.000, C 0.000 }
gfCNCPoint1[3537] = {X 279.7377, Y 12.1868, Z -1.3333, A 0.000, B 0.000, C 0.000 }
gfCNCPoint1[3538] = {X 279.8242, Y 11.2718, Z -1.3333, A 0.000, B 0.000, C 0.000 }
gfCNCPoint1[3539] = {X 280.0808, Y 10.3892, Z -1.3333, A 0.000, B 0.000, C 0.000 }
gfCNCPoint1[3540] = {X 280.5255, Y 9.5281, Z -1.3333, A 0.000, B 0.000, C 0.000 }
gfCNCPoint1[3541] = {X 281.1316, Y 8.7719, Z -1.3333, A 0.000, B 0.000, C 0.000 }
gfCNCPoint1[3542] = {X 281.8752, Y 8.1503, Z -1.3333, A 0.000, B 0.000, C 0.000 }
gfCNCPoint1[3543] = {X 282.7270, Y 7.6880, Z -1.3333, A 0.000, B 0.000, C 0.000 }
gfCNCPoint1[3544] = {X 283.6533, Y 7.4030, Z -1.3333, A 0.000, B 0.000, C 0.000 }
gfCNCPoint1[3545] = {X 284.6177, Y 7.3068, Z -1.3333, A 0.000, B 0.000, C 0.000 }
gfCNCPoint1[3546] = {X 291.0611, Y 7.3068, Z -1.3333, A 0.000, B 0.000, C 0.000 }
gfCNCPoint1[3547] = {X 292.0255, Y 7.4030, Z -1.3333, A 0.000, B 0.000, C 0.000 }
gfCNCPoint1[3548] = {X 292.9518, Y 7.6880, Z -1.3333, A 0.000, B 0.000, C 0.000 }
gfCNCPoint1[3549] = {X 293.8036, Y 8.1503, Z -1.3333, A 0.000, B 0.000, C 0.000 }
gfCNCPoint1[3550] = {X 294.5472, Y 8.7719, Z -1.3333, A 0.000, B 0.000, C 0.000 }
gfCNCPoint1[3551] = {X 295.1533, Y 9.5281, Z -1.3333, A 0.000, B 0.000, C 0.000 }
gfCNCPoint1[3552] = {X 295.5980, Y 10.3892, Z -1.3333, A 0.000, B 0.000, C 0.000 }
gfCNCPoint1[3553] = {X 295.8044, Y 11.0397, Z -1.3333, A 0.000, B 0.000, C 0.000 }
gfCNCPoint1[3554] = {X 295.9180, Y 11.7127, Z -1.3333, A 0.000, B 0.000, C 0.000 }
gfCNCPoint1[3555] = {X 295.9354, Y 11.9495, Z -1.3333, A 0.000, B 0.000, C 0.000 }
gfCNCPoint1[3556] = {X 295.9411, Y 12.1868, Z -1.3333, A 0.000, B 0.000, C 0.000 }
gfCNCPoint1[3557] = {X 295.9409, Y 13.0237, Z -1.3333, A 0.000, B 0.000, C 0.000 }
gfCNCPoint1[3558] = {X 295.9342, Y 13.2382, Z -1.3333, A 0.000, B 0.000, C 0.000 }
gfCNCPoint1[3559] = {X 295.9180, Y 13.4521, Z -1.3333, A 0.000, B 0.000, C 0.000 }
gfCNCPoint1[3560] = {X 298.3067, Y 13.6853, Z -1.3333, A 0.000, B 0.000, C 0.000 }
gfCNCPoint1[3561] = {X 298.1360, Y 14.6940, Z -1.3333, A 0.000, B 0.000, C 0.000 }
gfCNCPoint1[3562] = {X 297.8256, Y 15.6689, Z -1.3333, A 0.000, B 0.000, C 0.000 }
gfCNCPoint1[3563] = {X 297.3815, Y 16.5907, Z -1.3333, A 0.000, B 0.000, C 0.000 }
gfCNCPoint1[3564] = {X 296.8126, Y 17.4410, Z -1.3333, A 0.000, B 0.000, C 0.000 }
gfCNCPoint1[3565] = {X 296.8131, Y 19.2365, Z -1.3333, A 0.000, B 0.000, C 0.000 }
gfCNCPoint1[3566] = {X 299.8003, Y 19.2365, Z -1.3333, A 0.000, B 0.000, C 0.000 }
gfCNCPoint1[3567] = {X 299.8005, Y 17.4407, Z -1.3333, A 0.000, B 0.000, C 0.000 }
gfCNCPoint1[3568] = {X 299.2317, Y 16.5904, Z -1.3333, A 0.000, B 0.000, C 0.000 }
gfCNCPoint1[3569] = {X 298.7877, Y 15.6687, Z -1.3333, A 0.000, B 0.000, C 0.000 }
gfCNCPoint1[3570] = {X 298.4774, Y 14.6939, Z -1.3333, A 0.000, B 0.000, C 0.000 }
gfCNCPoint1[3571] = {X 298.3067, Y 13.6853, Z -1.3333, A 0.000, B 0.000, C 0.000 }
gfCNCPoint1[3572] = {X 295.9180, Y 13.4521, Z -1.3333, A 0.000, B 0.000, C 0.000 }
gfCNCPoint1[3573] = {X 295.7559, Y 14.3099, Z -1.3333, A 0.000, B 0.000, C 0.000 }
gfCNCPoint1[3574] = {X 295.4435, Y 15.1250, Z -1.3333, A 0.000, B 0.000, C 0.000 }
gfCNCPoint1[3575] = {X 294.9908, Y 15.8715, Z -1.3333, A 0.000, B 0.000, C 0.000 }
gfCNCPoint1[3576] = {X 294.4124, Y 16.5253, Z -1.3333, A 0.000, B 0.000, C 0.000 }
gfCNCPoint1[3577] = {X 294.4136, Y 21.6365, Z -1.3333, A 0.000, B 0.000, C 0.000 }
gfCNCPoint1[3578] = {X 302.2000, Y 21.6365, Z -1.3333, A 0.000, B 0.000, C 0.000 }
gfCNCPoint1[3579] = {X 302.2006, Y 16.5249, Z -1.3333, A 0.000, B 0.000, C 0.000 }
gfCNCPoint1[3580] = {X 301.6223, Y 15.8711, Z -1.3333, A 0.000, B 0.000, C 0.000 }
gfCNCPoint1[3581] = {X 301.1698, Y 15.1248, Z -1.3333, A 0.000, B 0.000, C 0.000 }
gfCNCPoint1[3582] = {X 300.8575, Y 14.3097, Z -1.3333, A 0.000, B 0.000, C 0.000 }
gfCNCPoint1[3583] = {X 300.6953, Y 13.4521, Z -1.3333, A 0.000, B 0.000, C 0.000 }
gfCNCPoint1[3584] = {X 300.6791, Y 13.2371, Z -1.3333, A 0.000, B 0.000, C 0.000 }
gfCNCPoint1[3585] = {X 300.6724, Y 13.0215, Z -1.3333, A 0.000, B 0.000, C 0.000 }
gfCNCPoint1[3586] = {X 300.6723, Y 12.1868, Z -1.3333, A 0.000, B 0.000, C 0.000 }
gfCNCPoint1[3587] = {X 300.6780, Y 11.9495, Z -1.3333, A 0.000, B 0.000, C 0.000 }
gfCNCPoint1[3588] = {X 300.6953, Y 11.7127, Z -1.3333, A 0.000, B 0.000, C 0.000 }
gfCNCPoint1[3589] = {X 300.8090, Y 11.0397, Z -1.3333, A 0.000, B 0.000, C 0.000 }
gfCNCPoint1[3590] = {X 301.0154, Y 10.3892, Z -1.3333, A 0.000, B 0.000, C 0.000 }
gfCNCPoint1[3591] = {X 301.4601, Y 9.5281, Z -1.3333, A 0.000, B 0.000, C 0.000 }
gfCNCPoint1[3592] = {X 302.0662, Y 8.7719, Z -1.3333, A 0.000, B 0.000, C 0.000 }
gfCNCPoint1[3593] = {X 302.8098, Y 8.1503, Z -1.3333, A 0.000, B 0.000, C 0.000 }
gfCNCPoint1[3594] = {X 303.6616, Y 7.6880, Z -1.3333, A 0.000, B 0.000, C 0.000 }
gfCNCPoint1[3595] = {X 304.5879, Y 7.4030, Z -1.3333, A 0.000, B 0.000, C 0.000 }
gfCNCPoint1[3596] = {X 305.5523, Y 7.3068, Z -1.3333, A 0.000, B 0.000, C 0.000 }
gfCNCPoint1[3597] = {X 311.9957, Y 7.3068, Z -1.3333, A 0.000, B 0.000, C 0.000 }
gfCNCPoint1[3598] = {X 312.9478, Y 7.4006, Z -1.3333, A 0.000, B 0.000, C 0.000 }
gfCNCPoint1[3599] = {X 313.8632, Y 7.6783, Z -1.3333, A 0.000, B 0.000, C 0.000 }
gfCNCPoint1[3600] = {X 314.7069, Y 8.1292, Z -1.3333, A 0.000, B 0.000, C 0.000 }
gfCNCPoint1[3601] = {X 315.4464, Y 8.7361, Z -1.3333, A 0.000, B 0.000, C 0.000 }
gfCNCPoint1[3602] = {X 316.0533, Y 9.4756, Z -1.3333, A 0.000, B 0.000, C 0.000 }
gfCNCPoint1[3603] = {X 316.5043, Y 10.3193, Z -1.3333, A 0.000, B 0.000, C 0.000 }
gfCNCPoint1[3604] = {X 316.7820, Y 11.2348, Z -1.3333, A 0.000, B 0.000, C 0.000 }
gfCNCPoint1[3605] = {X 316.8757, Y 12.1868, Z -1.3333, A 0.000, B 0.000, C 0.000 }
gfCNCPoint1[3606] = {X 316.8755, Y 13.0237, Z -1.3333, A 0.000, B 0.000, C 0.000 }
gfCNCPoint1[3607] = {X 316.7680, Y 13.9975, Z -1.3333, A 0.000, B 0.000, C 0.000 }
gfCNCPoint1[3608] = {X 316.4682, Y 14.9302, Z -1.3333, A 0.000, B 0.000, C 0.000 }
gfCNCPoint1[3609] = {X 315.9881, Y 15.7843, Z -1.3333, A 0.000, B 0.000, C 0.000 }
gfCNCPoint1[3610] = {X 315.3471, Y 16.5252, Z -1.3333, A 0.000, B 0.000, C 0.000 }
gfCNCPoint1[3611] = {X 315.3469, Y 40.6614, Z -1.3333, A 0.000, B 0.000, C 0.000 }
gfCNCPoint1[3612] = {X 315.9885, Y 41.4030, Z -1.3333, A 0.000, B 0.000, C 0.000 }
gfCNCPoint1[3613] = {X 316.4688, Y 42.2579, Z -1.3333, A 0.000, B 0.000, C 0.000 }
gfCNCPoint1[3614] = {X 316.7685, Y 43.1916, Z -1.3333, A 0.000, B 0.000, C 0.000 }
gfCNCPoint1[3615] = {X 316.8755, Y 44.1664, Z -1.3333, A 0.000, B 0.000, C 0.000 }
gfCNCPoint1[3616] = {X 316.8757, Y 45.0000, Z -1.3333, A 0.000, B 0.000, C 0.000 }
gfCNCPoint1[3617] = {X 316.8749, Y 45.0899, Z -1.3333, A 0.000, B 0.000, C 0.000 }
gfCNCPoint1[3618] = {X 316.8724, Y 45.1799, Z -1.3333, A 0.000, B 0.000, C 0.000 }
gfCNCPoint1[3619] = {X 316.8594, Y 45.3987, Z -1.3333, A 0.000, B 0.000, C 0.000 }
gfCNCPoint1[3620] = {X 316.8366, Y 45.6167, Z -1.3333, A 0.000, B 0.000, C 0.000 }
gfCNCPoint1[3621] = {X 316.6062, Y 46.5992, Z -1.3333, A 0.000, B 0.000, C 0.000 }
gfCNCPoint1[3622] = {X 316.1787, Y 47.5134, Z -1.3333, A 0.000, B 0.000, C 0.000 }
gfCNCPoint1[3623] = {X 315.5723, Y 48.3200, Z -1.3333, A 0.000, B 0.000, C 0.000 }
gfCNCPoint1[3624] = {X 315.2205, Y 47.9934, Z -1.3333, A 0.000, B 0.000, C 0.000 }
gfCNCPoint1[3625] = {X 314.5413, Y 48.5889, Z -1.3333, A 0.000, B 0.000, C 0.000 }
gfCNCPoint1[3626] = {X 313.7548, Y 49.0331, Z -1.3333, A 0.000, B 0.000, C 0.000 }
gfCNCPoint1[3627] = {X 312.8942, Y 49.3073, Z -1.3333, A 0.000, B 0.000, C 0.000 }
gfCNCPoint1[3628] = {X 311.9957, Y 49.4000, Z -1.3333, A 0.000, B 0.000, C 0.000 }
gfCNCPoint1[3629] = {X 305.5523, Y 49.4000, Z -1.3333, A 0.000, B 0.000, C 0.000 }
gfCNCPoint1[3630] = {X 304.5732, Y 49.2897, Z -1.3333, A 0.000, B 0.000, C 0.000 }
gfCNCPoint1[3631] = {X 303.6432, Y 48.9643, Z -1.3333, A 0.000, B 0.000, C 0.000 }
gfCNCPoint1[3632] = {X 302.8089, Y 48.4400, Z -1.3333, A 0.000, B 0.000, C 0.000 }
